// @TEST-RUN
converted := TryConvert_UDINT_TO_Destination(value, actual);
equal := actual = UDINT_TO_BOOL(value);

// @TEST-ASSERT
AssertTrue(Condition := equal, Message := 'Did not convert UDINT to BOOL correctly');
AssertTrue(Condition := converted, Message := 'Did not report UDINT to BOOL conversion was successful');

TEST_FINISHED();
END_METHOD

METHOD PUBLIC Check_UDINT_TO_BOOL_Max
VAR
	value : UDINT := DatatypeLimits.UDINT_MAX_VALUE;
	actual : BOOL;
	converted : BOOL;
	equal : BOOL;
END_VAR
TEST('Check_UDINT_TO_BOOL_Max');

// @TEST-RUN
converted := TryConvert_UDINT_TO_Destination(value, actual);
equal := actual = UDINT_TO_BOOL(value);

// @TEST-ASSERT
AssertTrue(Condition := equal, Message := 'Did not convert UDINT to BOOL correctly');
AssertTrue(Condition := converted, Message := 'Did not report UDINT to BOOL conversion was successful');

TEST_FINISHED();
END_METHOD

METHOD PUBLIC Check_UDINT_TO_BYTE_Min
VAR
	value : UDINT := DatatypeLimits.UDINT_MIN_VALUE;
	actual : BYTE;
	converted : BOOL;
	equal : BOOL;
END_VAR
TEST('Check_UDINT_TO_BYTE_Min');

// @TEST-RUN
converted := TryConvert_UDINT_TO_Destination(value, actual);
equal := actual = UDINT_TO_BYTE(value);

// @TEST-ASSERT
AssertTrue(Condition := equal, Message := 'Did not convert UDINT to BYTE correctly');
AssertTrue(Condition := converted, Message := 'Did not report UDINT to BYTE conversion was successful');

TEST_FINISHED();
END_METHOD

METHOD PUBLIC Check_UDINT_TO_BYTE_TooHigh
VAR
	value : UDINT := DatatypeLimits.UDINT_MAX_VALUE;
	actual : BYTE;
	converted : BOOL;
END_VAR
TEST('Check_UDINT_TO_BYTE_TooHigh');

// @TEST-RUN
converted := TryConvert_UDINT_TO_Destination(value, actual);

// @TEST-ASSERT
AssertFalse(Condition := converted, Message := 'Did not report UDINT to BYTE conversion was prevented');

TEST_FINISHED();
END_METHOD

METHOD PUBLIC Check_UDINT_TO_BYTE_Max
VAR
	value : UDINT := DatatypeLimits.MAX_VALUE_OF_UDINT_WHICH_CAN_BE_HELD_IN_A_BYTE;
	actual : BYTE;
	converted : BOOL;
	equal : BOOL;
END_VAR
TEST('Check_UDINT_TO_BYTE_Max');

// @TEST-RUN
converted := TryConvert_UDINT_TO_Destination(value, actual);
equal := actual = UDINT_TO_BYTE(value);

// @TEST-ASSERT
AssertTrue(Condition := equal, Message := 'Did not convert UDINT to BYTE correctly');
AssertTrue(Condition := converted, Message := 'Did not report UDINT to BYTE conversion was successful');

TEST_FINISHED();
END_METHOD

METHOD PUBLIC Check_UDINT_TO_DATE_Min
VAR
	value : UDINT := DatatypeLimits.UDINT_MIN_VALUE;
	actual : DATE;
	converted : BOOL;
	equal : BOOL;
END_VAR
TEST('Check_UDINT_TO_DATE_Min');

// @TEST-RUN
converted := TryConvert_UDINT_TO_Destination(value, actual);
equal := actual = UDINT_TO_DATE(value);

// @TEST-ASSERT
AssertTrue(Condition := equal, Message := 'Did not convert UDINT to DATE correctly');
AssertTrue(Condition := converted, Message := 'Did not report UDINT to DATE conversion was successful');

TEST_FINISHED();
END_METHOD

METHOD PUBLIC Check_UDINT_TO_DATE_Max
VAR
	value : UDINT := DatatypeLimits.UDINT_MAX_VALUE;
	actual : DATE;
	converted : BOOL;
	equal : BOOL;
END_VAR
TEST('Check_UDINT_TO_DATE_Max');

// @TEST-RUN
converted := TryConvert_UDINT_TO_Destination(value, actual);
equal := actual = UDINT_TO_DATE(value);

// @TEST-ASSERT
AssertTrue(Condition := equal, Message := 'Did not convert UDINT to DATE correctly');
AssertTrue(Condition := converted, Message := 'Did not report UDINT to DATE conversion was successful');

TEST_FINISHED();
END_METHOD

METHOD PUBLIC Check_UDINT_TO_DINT_Min
VAR
	value : UDINT := DatatypeLimits.UDINT_MIN_VALUE;
	actual : DINT;
	converted : BOOL;
	equal : BOOL;
END_VAR
TEST('Check_UDINT_TO_DINT_Min');

// @TEST-RUN
converted := TryConvert_UDINT_TO_Destination(value, actual);
equal := actual = UDINT_TO_DINT(value);

// @TEST-ASSERT
AssertTrue(Condition := equal, Message := 'Did not convert UDINT to DINT correctly');
AssertTrue(Condition := converted, Message := 'Did not report UDINT to DINT conversion was successful');

TEST_FINISHED();
END_METHOD

METHOD PUBLIC Check_UDINT_TO_DINT_TooHigh
VAR
	value : UDINT := DatatypeLimits.UDINT_MAX_VALUE;
	actual : DINT;
	converted : BOOL;
END_VAR
TEST('Check_UDINT_TO_DINT_TooHigh');

// @TEST-RUN
converted := TryConvert_UDINT_TO_Destination(value, actual);

// @TEST-ASSERT
AssertFalse(Condition := converted, Message := 'Did not report UDINT to DINT conversion was prevented');

TEST_FINISHED();
END_METHOD

METHOD PUBLIC Check_UDINT_TO_DINT_Max
VAR
	value : UDINT := DatatypeLimits.MAX_VALUE_OF_UDINT_WHICH_CAN_BE_HELD_IN_A_DINT;
	actual : DINT;
	converted : BOOL;
	equal : BOOL;
END_VAR
TEST('Check_UDINT_TO_DINT_Max');

// @TEST-RUN
converted := TryConvert_UDINT_TO_Destination(value, actual);
equal := actual = UDINT_TO_DINT(value);

// @TEST-ASSERT
AssertTrue(Condition := equal, Message := 'Did not convert UDINT to DINT correctly');
AssertTrue(Condition := converted, Message := 'Did not report UDINT to DINT conversion was successful');

TEST_FINISHED();
END_METHOD

METHOD PUBLIC Check_UDINT_TO_DT_Min
VAR
	value : UDINT := DatatypeLimits.UDINT_MIN_VALUE;
	actual : DT;
	converted : BOOL;
	equal : BOOL;
END_VAR
TEST('Check_UDINT_TO_DT_Min');

// @TEST-RUN
converted := TryConvert_UDINT_TO_Destination(value, actual);
equal := actual = UDINT_TO_DT(value);

// @TEST-ASSERT
AssertTrue(Condition := equal, Message := 'Did not convert UDINT to DT correctly');
AssertTrue(Condition := converted, Message := 'Did not report UDINT to DT conversion was successful');

TEST_FINISHED();
END_METHOD

METHOD PUBLIC Check_UDINT_TO_DT_Max
VAR
	value : UDINT := DatatypeLimits.UDINT_MAX_VALUE;
	actual : DT;
	converted : BOOL;
	equal : BOOL;
END_VAR
TEST('Check_UDINT_TO_DT_Max');

// @TEST-RUN
converted := TryConvert_UDINT_TO_Destination(value, actual);
equal := actual = UDINT_TO_DT(value);

// @TEST-ASSERT
AssertTrue(Condition := equal, Message := 'Did not convert UDINT to DT correctly');
AssertTrue(Condition := converted, Message := 'Did not report UDINT to DT conversion was successful');

TEST_FINISHED();
END_METHOD

METHOD PUBLIC Check_UDINT_TO_DWORD_Min
VAR
	value : UDINT := DatatypeLimits.UDINT_MIN_VALUE;
	actual : DWORD;
	converted : BOOL;
	equal : BOOL;
END_VAR
TEST('Check_UDINT_TO_DWORD_Min');

// @TEST-RUN
converted := TryConvert_UDINT_TO_Destination(value, actual);
equal := actual = UDINT_TO_DWORD(value);

// @TEST-ASSERT
AssertTrue(Condition := equal, Message := 'Did not convert UDINT to DWORD correctly');
AssertTrue(Condition := converted, Message := 'Did not report UDINT to DWORD conversion was successful');

TEST_FINISHED();
END_METHOD

METHOD PUBLIC Check_UDINT_TO_DWORD_Max
VAR
	value : UDINT := DatatypeLimits.UDINT_MAX_VALUE;
	actual : DWORD;
	converted : BOOL;
	equal : BOOL;
END_VAR
TEST('Check_UDINT_TO_DWORD_Max');

// @TEST-RUN
converted := TryConvert_UDINT_TO_Destination(value, actual);
equal := actual = UDINT_TO_DWORD(value);

// @TEST-ASSERT
AssertTrue(Condition := equal, Message := 'Did not convert UDINT to DWORD correctly');
AssertTrue(Condition := converted, Message := 'Did not report UDINT to DWORD conversion was successful');

TEST_FINISHED();
END_METHOD

METHOD PUBLIC Check_UDINT_TO_INT_Min
VAR
	value : UDINT := DatatypeLimits.UDINT_MIN_VALUE;
	actual : INT;
	converted : BOOL;
	equal : BOOL;
END_VAR
TEST('Check_UDINT_TO_INT_Min');

// @TEST-RUN
converted := TryConvert_UDINT_TO_Destination(value, actual);
equal := actual = UDINT_TO_INT(value);

// @TEST-ASSERT
AssertTrue(Condition := equal, Message := 'Did not convert UDINT to INT correctly');
AssertTrue(Condition := converted, Message := 'Did not report UDINT to INT conversion was successful');

TEST_FINISHED();
END_METHOD

METHOD PUBLIC Check_UDINT_TO_INT_TooHigh
VAR
	value : UDINT := DatatypeLimits.UDINT_MAX_VALUE;
	actual : INT;
	converted : BOOL;
END_VAR
TEST('Check_UDINT_TO_INT_TooHigh');

// @TEST-RUN
converted := TryConvert_UDINT_TO_Destination(value, actual);

// @TEST-ASSERT
AssertFalse(Condition := converted, Message := 'Did not report UDINT to INT conversion was prevented');

TEST_FINISHED();
END_METHOD

METHOD PUBLIC Check_UDINT_TO_INT_Max
VAR
	value : UDINT := DatatypeLimits.MAX_VALUE_OF_UDINT_WHICH_CAN_BE_HELD_IN_A_INT;
	actual : INT;
	converted : BOOL;
	equal : BOOL;
END_VAR
TEST('Check_UDINT_TO_INT_Max');

// @TEST-RUN
converted := TryConvert_UDINT_TO_Destination(value, actual);
equal := actual = UDINT_TO_INT(value);

// @TEST-ASSERT
AssertTrue(Condition := equal, Message := 'Did not convert UDINT to INT correctly');
AssertTrue(Condition := converted, Message := 'Did not report UDINT to INT conversion was successful');

TEST_FINISHED();
END_METHOD

METHOD PUBLIC Check_UDINT_TO_LINT_Min
VAR
	value : UDINT := DatatypeLimits.UDINT_MIN_VALUE;
	actual : LINT;
	converted : BOOL;
	equal : BOOL;
END_VAR
TEST('Check_UDINT_TO_LINT_Min');

// @TEST-RUN
converted := TryConvert_UDINT_TO_Destination(value, actual);
equal := actual = UDINT_TO_LINT(value);

// @TEST-ASSERT
AssertTrue(Condition := equal, Message := 'Did not convert UDINT to LINT correctly');
AssertTrue(Condition := converted, Message := 'Did not report UDINT to LINT conversion was successful');

TEST_FINISHED();
END_METHOD

METHOD PUBLIC Check_UDINT_TO_LINT_Max
VAR
	value : UDINT := DatatypeLimits.UDINT_MAX_VALUE;
	actual : LINT;
	converted : BOOL;
	equal : BOOL;
END_VAR
TEST('Check_UDINT_TO_LINT_Max');

// @TEST-RUN
converted := TryConvert_UDINT_TO_Destination(value, actual);
equal := actual = UDINT_TO_LINT(value);

// @TEST-ASSERT
AssertTrue(Condition := equal, Message := 'Did not convert UDINT to LINT correctly');
AssertTrue(Condition := converted, Message := 'Did not report UDINT to LINT conversion was successful');

TEST_FINISHED();
END_METHOD

METHOD PUBLIC Check_UDINT_TO_LREAL_Min
VAR
	value : UDINT := DatatypeLimits.UDINT_MIN_VALUE;
	actual : LREAL;
	converted : BOOL;
	equal : BOOL;
END_VAR
TEST('Check_UDINT_TO_LREAL_Min');

// @TEST-RUN
converted := TryConvert_UDINT_TO_Destination(value, actual);
equal := actual = UDINT_TO_LREAL(value);

// @TEST-ASSERT
AssertTrue(Condition := equal, Message := 'Did not convert UDINT to LREAL correctly');
AssertTrue(Condition := converted, Message := 'Did not report UDINT to LREAL conversion was successful');

TEST_FINISHED();
END_METHOD

METHOD PUBLIC Check_UDINT_TO_LREAL_Max
VAR
	value : UDINT := DatatypeLimits.UDINT_MAX_VALUE;
	actual : LREAL;
	converted : BOOL;
	equal : BOOL;
END_VAR
TEST('Check_UDINT_TO_LREAL_Max');

// @TEST-RUN
converted := TryConvert_UDINT_TO_Destination(value, actual);
equal := actual = UDINT_TO_LREAL(value);

// @TEST-ASSERT
AssertTrue(Condition := equal, Message := 'Did not convert UDINT to LREAL correctly');
AssertTrue(Condition := converted, Message := 'Did not report UDINT to LREAL conversion was successful');

TEST_FINISHED();
END_METHOD

METHOD PUBLIC Check_UDINT_TO_LWORD_Min
VAR
	value : UDINT := DatatypeLimits.UDINT_MIN_VALUE;
	actual : LWORD;
	converted : BOOL;
	equal : BOOL;
END_VAR
TEST('Check_UDINT_TO_LWORD_Min');

// @TEST-RUN
converted := TryConvert_UDINT_TO_Destination(value, actual);
equal := actual = UDINT_TO_LWORD(value);

// @TEST-ASSERT
AssertTrue(Condition := equal, Message := 'Did not convert UDINT to LWORD correctly');
AssertTrue(Condition := converted, Message := 'Did not report UDINT to LWORD conversion was successful');

TEST_FINISHED();
END_METHOD

METHOD PUBLIC Check_UDINT_TO_LWORD_Max
VAR
	value : UDINT := DatatypeLimits.UDINT_MAX_VALUE;
	actual : LWORD;
	converted : BOOL;
	equal : BOOL;
END_VAR
TEST('Check_UDINT_TO_LWORD_Max');

// @TEST-RUN
converted := TryConvert_UDINT_TO_Destination(value, actual);
equal := actual = UDINT_TO_LWORD(value);

// @TEST-ASSERT
AssertTrue(Condition := equal, Message := 'Did not convert UDINT to LWORD correctly');
AssertTrue(Condition := converted, Message := 'Did not report UDINT to LWORD conversion was successful');

TEST_FINISHED();
END_METHOD

METHOD PUBLIC Check_UDINT_TO_REAL_Min
VAR
	value : UDINT := DatatypeLimits.UDINT_MIN_VALUE;
	actual : REAL;
	converted : BOOL;
	equal : BOOL;
END_VAR
TEST('Check_UDINT_TO_REAL_Min');

// @TEST-RUN
converted := TryConvert_UDINT_TO_Destination(value, actual);
equal := actual = UDINT_TO_REAL(value);

// @TEST-ASSERT
AssertTrue(Condition := equal, Message := 'Did not convert UDINT to REAL correctly');
AssertTrue(Condition := converted, Message := 'Did not report UDINT to REAL conversion was successful');

TEST_FINISHED();
END_METHOD

METHOD PUBLIC Check_UDINT_TO_REAL_Max
VAR
	value : UDINT := DatatypeLimits.UDINT_MAX_VALUE;
	actual : REAL;
	converted : BOOL;
	equal : BOOL;
END_VAR
TEST('Check_UDINT_TO_REAL_Max');

// @TEST-RUN
converted := TryConvert_UDINT_TO_Destination(value, actual);
equal := actual = UDINT_TO_REAL(value);

// @TEST-ASSERT
AssertTrue(Condition := equal, Message := 'Did not convert UDINT to REAL correctly');
AssertTrue(Condition := converted, Message := 'Did not report UDINT to REAL conversion was successful');

TEST_FINISHED();
END_METHOD

METHOD PUBLIC Check_UDINT_TO_SINT_Min
VAR
	value : UDINT := DatatypeLimits.UDINT_MIN_VALUE;
	actual : SINT;
	converted : BOOL;
	equal : BOOL;
END_VAR
TEST('Check_UDINT_TO_SINT_Min');

// @TEST-RUN
converted := TryConvert_UDINT_TO_Destination(value, actual);
equal := actual = UDINT_TO_SINT(value);

// @TEST-ASSERT
AssertTrue(Condition := equal, Message := 'Did not convert UDINT to SINT correctly');
AssertTrue(Condition := converted, Message := 'Did not report UDINT to SINT conversion was successful');

TEST_FINISHED();
END_METHOD

METHOD PUBLIC Check_UDINT_TO_SINT_TooHigh
VAR
	value : UDINT := DatatypeLimits.UDINT_MAX_VALUE;
	actual : SINT;
	converted : BOOL;
END_VAR
TEST('Check_UDINT_TO_SINT_TooHigh');

// @TEST-RUN
converted := TryConvert_UDINT_TO_Destination(value, actual);

// @TEST-ASSERT
AssertFalse(Condition := converted, Message := 'Did not report UDINT to SINT conversion was prevented');

TEST_FINISHED();
END_METHOD

METHOD PUBLIC Check_UDINT_TO_SINT_Max
VAR
	value : UDINT := DatatypeLimits.MAX_VALUE_OF_UDINT_WHICH_CAN_BE_HELD_IN_A_SINT;
	actual : SINT;
	converted : BOOL;
	equal : BOOL;
END_VAR
TEST('Check_UDINT_TO_SINT_Max');

// @TEST-RUN
converted := TryConvert_UDINT_TO_Destination(value, actual);
equal := actual = UDINT_TO_SINT(value);

// @TEST-ASSERT
AssertTrue(Condition := equal, Message := 'Did not convert UDINT to SINT correctly');
AssertTrue(Condition := converted, Message := 'Did not report UDINT to SINT conversion was successful');

TEST_FINISHED();
END_METHOD

METHOD PUBLIC Check_UDINT_TO_STRING_Min
VAR
	value : UDINT := DatatypeLimits.UDINT_MIN_VALUE;
	actual : STRING;
	converted : BOOL;
	equal : BOOL;
END_VAR
TEST('Check_UDINT_TO_STRING_Min');

// @TEST-RUN
converted := TryConvert_UDINT_TO_Destination(value, actual);
equal := actual = UDINT_TO_STRING(value);

// @TEST-ASSERT
AssertTrue(Condition := equal, Message := 'Did not convert UDINT to STRING correctly');
AssertTrue(Condition := converted, Message := 'Did not report UDINT to STRING conversion was successful');

TEST_FINISHED();
END_METHOD

METHOD PUBLIC Check_UDINT_TO_STRING_Max
VAR
	value : UDINT := DatatypeLimits.UDINT_MAX_VALUE;
	actual : STRING;
	converted : BOOL;
	equal : BOOL;
END_VAR
TEST('Check_UDINT_TO_STRING_Max');

// @TEST-RUN
converted := TryConvert_UDINT_TO_Destination(value, actual);
equal := actual = UDINT_TO_STRING(value);

// @TEST-ASSERT
AssertTrue(Condition := equal, Message := 'Did not convert UDINT to STRING correctly');
AssertTrue(Condition := converted, Message := 'Did not report UDINT to STRING conversion was successful');

TEST_FINISHED();
END_METHOD

METHOD PUBLIC Check_UDINT_TO_TIME_Min
VAR
	value : UDINT := DatatypeLimits.UDINT_MIN_VALUE;
	actual : TIME;
	converted : BOOL;
	equal : BOOL;
END_VAR
TEST('Check_UDINT_TO_TIME_Min');

// @TEST-RUN
converted := TryConvert_UDINT_TO_Destination(value, actual);
equal := actual = UDINT_TO_TIME(value);

// @TEST-ASSERT
AssertTrue(Condition := equal, Message := 'Did not convert UDINT to TIME correctly');
AssertTrue(Condition := converted, Message := 'Did not report UDINT to TIME conversion was successful');

TEST_FINISHED();
END_METHOD

METHOD PUBLIC Check_UDINT_TO_TIME_Max
VAR
	value : UDINT := DatatypeLimits.UDINT_MAX_VALUE;
	actual : TIME;
	converted : BOOL;
	equal : BOOL;
END_VAR
TEST('Check_UDINT_TO_TIME_Max');

// @TEST-RUN
converted := TryConvert_UDINT_TO_Destination(value, actual);
equal := actual = UDINT_TO_TIME(value);

// @TEST-ASSERT
AssertTrue(Condition := equal, Message := 'Did not convert UDINT to TIME correctly');
AssertTrue(Condition := converted, Message := 'Did not report UDINT to TIME conversion was successful');

TEST_FINISHED();
END_METHOD

METHOD PUBLIC Check_UDINT_TO_TOD_Min
VAR
	value : UDINT := DatatypeLimits.UDINT_MIN_VALUE;
	actual : TOD;
	converted : BOOL;
	equal : BOOL;
END_VAR
TEST('Check_UDINT_TO_TOD_Min');

// @TEST-RUN
converted := TryConvert_UDINT_TO_Destination(value, actual);
equal := actual = UDINT_TO_TOD(value);

// @TEST-ASSERT
AssertTrue(Condition := equal, Message := 'Did not convert UDINT to TOD correctly');
AssertTrue(Condition := converted, Message := 'Did not report UDINT to TOD conversion was successful');

TEST_FINISHED();
END_METHOD

METHOD PUBLIC Check_UDINT_TO_TOD_TooHigh
VAR
	value : UDINT := DatatypeLimits.UDINT_MAX_VALUE;
	actual : TOD;
	converted : BOOL;
END_VAR
TEST('Check_UDINT_TO_TOD_TooHigh');

// @TEST-RUN
converted := TryConvert_UDINT_TO_Destination(value, actual);

// @TEST-ASSERT
AssertFalse(Condition := converted, Message := 'Did not report UDINT to TOD conversion was prevented');

TEST_FINISHED();
END_METHOD

METHOD PUBLIC Check_UDINT_TO_TOD_Max
VAR
	value : UDINT := DatatypeLimits.MAX_VALUE_OF_UDINT_WHICH_CAN_BE_HELD_IN_A_TOD;
	actual : TOD;
	converted : BOOL;
	equal : BOOL;
END_VAR
TEST('Check_UDINT_TO_TOD_Max');

// @TEST-RUN
converted := TryConvert_UDINT_TO_Destination(value, actual);
equal := actual = UDINT_TO_TOD(value);

// @TEST-ASSERT
AssertTrue(Condition := equal, Message := 'Did not convert UDINT to TOD correctly');
AssertTrue(Condition := converted, Message := 'Did not report UDINT to TOD conversion was successful');

TEST_FINISHED();
END_METHOD

METHOD PUBLIC Check_UDINT_TO_UDINT_Min
VAR
	value : UDINT := DatatypeLimits.UDINT_MIN_VALUE;
	actual : UDINT;
	converted : BOOL;
	equal : BOOL;
END_VAR
TEST('Check_UDINT_TO_UDINT_Min');

// @TEST-RUN
converted := TryConvert_UDINT_TO_Destination(value, actual);
equal := actual = value;

// @TEST-ASSERT
AssertTrue(Condition := equal, Message := 'Did not convert UDINT to UDINT correctly');
AssertTrue(Condition := converted, Message := 'Did not report UDINT to UDINT conversion was successful');

TEST_FINISHED();
END_METHOD

METHOD PUBLIC Check_UDINT_TO_UDINT_Max
VAR
	value : UDINT := DatatypeLimits.UDINT_MAX_VALUE;
	actual : UDINT;
	converted : BOOL;
	equal : BOOL;
END_VAR
TEST('Check_UDINT_TO_UDINT_Max');

// @TEST-RUN
converted := TryConvert_UDINT_TO_Destination(value, actual);
equal := actual = value;

// @TEST-ASSERT
AssertTrue(Condition := equal, Message := 'Did not convert UDINT to UDINT correctly');
AssertTrue(Condition := converted, Message := 'Did not report UDINT to UDINT conversion was successful');

TEST_FINISHED();
END_METHOD

METHOD PUBLIC Check_UDINT_TO_UINT_Min
VAR
	value : UDINT := DatatypeLimits.UDINT_MIN_VALUE;
	actual : UINT;
	converted : BOOL;
	equal : BOOL;
END_VAR
TEST('Check_UDINT_TO_UINT_Min');

// @TEST-RUN
converted := TryConvert_UDINT_TO_Destination(value, actual);
equal := actual = UDINT_TO_UINT(value);

// @TEST-ASSERT
AssertTrue(Condition := equal, Message := 'Did not convert UDINT to UINT correctly');
AssertTrue(Condition := converted, Message := 'Did not report UDINT to UINT conversion was successful');

TEST_FINISHED();
END_METHOD

METHOD PUBLIC Check_UDINT_TO_UINT_TooHigh
VAR
	value : UDINT := DatatypeLimits.UDINT_MAX_VALUE;
	actual : UINT;
	converted : BOOL;
END_VAR
TEST('Check_UDINT_TO_UINT_TooHigh');

// @TEST-RUN
converted := TryConvert_UDINT_TO_Destination(value, actual);

// @TEST-ASSERT
AssertFalse(Condition := converted, Message := 'Did not report UDINT to UINT conversion was prevented');

TEST_FINISHED();
END_METHOD

METHOD PUBLIC Check_UDINT_TO_UINT_Max
VAR
	value : UDINT := DatatypeLimits.MAX_VALUE_OF_UDINT_WHICH_CAN_BE_HELD_IN_A_UINT;
	actual : UINT;
	converted : BOOL;
	equal : BOOL;
END_VAR
TEST('Check_UDINT_TO_UINT_Max');

// @TEST-RUN
converted := TryConvert_UDINT_TO_Destination(value, actual);
equal := actual = UDINT_TO_UINT(value);

// @TEST-ASSERT
AssertTrue(Condition := equal, Message := 'Did not convert UDINT to UINT correctly');
AssertTrue(Condition := converted, Message := 'Did not report UDINT to UINT conversion was successful');

TEST_FINISHED();
END_METHOD

METHOD PUBLIC Check_UDINT_TO_ULINT_Min
VAR
	value : UDINT := DatatypeLimits.UDINT_MIN_VALUE;
	actual : ULINT;
	converted : BOOL;
	equal : BOOL;
END_VAR
TEST('Check_UDINT_TO_ULINT_Min');

// @TEST-RUN
converted := TryConvert_UDINT_TO_Destination(value, actual);
equal := actual = UDINT_TO_ULINT(value);

// @TEST-ASSERT
AssertTrue(Condition := equal, Message := 'Did not convert UDINT to ULINT correctly');
AssertTrue(Condition := converted, Message := 'Did not report UDINT to ULINT conversion was successful');

TEST_FINISHED();
END_METHOD

METHOD PUBLIC Check_UDINT_TO_ULINT_Max
VAR
	value : UDINT := DatatypeLimits.UDINT_MAX_VALUE;
	actual : ULINT;
	converted : BOOL;
	equal : BOOL;
END_VAR
TEST('Check_UDINT_TO_ULINT_Max');

// @TEST-RUN
converted := TryConvert_UDINT_TO_Destination(value, actual);
equal := actual = UDINT_TO_ULINT(value);

// @TEST-ASSERT
AssertTrue(Condition := equal, Message := 'Did not convert UDINT to ULINT correctly');
AssertTrue(Condition := converted, Message := 'Did not report UDINT to ULINT conversion was successful');

TEST_FINISHED();
END_METHOD

METHOD PUBLIC Check_UDINT_TO_USINT_Min
VAR
	value : UDINT := DatatypeLimits.UDINT_MIN_VALUE;
	actual : USINT;
	converted : BOOL;
	equal : BOOL;
END_VAR
TEST('Check_UDINT_TO_USINT_Min');

// @TEST-RUN
converted := TryConvert_UDINT_TO_Destination(value, actual);
equal := actual = UDINT_TO_USINT(value);

// @TEST-ASSERT
AssertTrue(Condition := equal, Message := 'Did not convert UDINT to USINT correctly');
AssertTrue(Condition := converted, Message := 'Did not report UDINT to USINT conversion was successful');

TEST_FINISHED();
END_METHOD

METHOD PUBLIC Check_UDINT_TO_USINT_TooHigh
VAR
	value : UDINT := DatatypeLimits.UDINT_MAX_VALUE;
	actual : USINT;
	converted : BOOL;
END_VAR
TEST('Check_UDINT_TO_USINT_TooHigh');

// @TEST-RUN
converted := TryConvert_UDINT_TO_Destination(value, actual);

// @TEST-ASSERT
AssertFalse(Condition := converted, Message := 'Did not report UDINT to USINT conversion was prevented');

TEST_FINISHED();
END_METHOD

METHOD PUBLIC Check_UDINT_TO_USINT_Max
VAR
	value : UDINT := DatatypeLimits.MAX_VALUE_OF_UDINT_WHICH_CAN_BE_HELD_IN_A_USINT;
	actual : USINT;
	converted : BOOL;
	equal : BOOL;
END_VAR
TEST('Check_UDINT_TO_USINT_Max');

// @TEST-RUN
converted := TryConvert_UDINT_TO_Destination(value, actual);
equal := actual = UDINT_TO_USINT(value);

// @TEST-ASSERT
AssertTrue(Condition := equal, Message := 'Did not convert UDINT to USINT correctly');
AssertTrue(Condition := converted, Message := 'Did not report UDINT to USINT conversion was successful');

TEST_FINISHED();
END_METHOD

METHOD PUBLIC Check_UDINT_TO_WORD_Min
VAR
	value : UDINT := DatatypeLimits.UDINT_MIN_VALUE;
	actual : WORD;
	converted : BOOL;
	equal : BOOL;
END_VAR
TEST('Check_UDINT_TO_WORD_Min');

// @TEST-RUN
converted := TryConvert_UDINT_TO_Destination(value, actual);
equal := actual = UDINT_TO_WORD(value);

// @TEST-ASSERT
AssertTrue(Condition := equal, Message := 'Did not convert UDINT to WORD correctly');
AssertTrue(Condition := converted, Message := 'Did not report UDINT to WORD conversion was successful');

TEST_FINISHED();
END_METHOD

METHOD PUBLIC Check_UDINT_TO_WORD_TooHigh
VAR
	value : UDINT := DatatypeLimits.UDINT_MAX_VALUE;
	actual : WORD;
	converted : BOOL;
END_VAR
TEST('Check_UDINT_TO_WORD_TooHigh');

// @TEST-RUN
converted := TryConvert_UDINT_TO_Destination(value, actual);

// @TEST-ASSERT
AssertFalse(Condition := converted, Message := 'Did not report UDINT to WORD conversion was prevented');

TEST_FINISHED();
END_METHOD

METHOD PUBLIC Check_UDINT_TO_WORD_Max
VAR
	value : UDINT := DatatypeLimits.MAX_VALUE_OF_UDINT_WHICH_CAN_BE_HELD_IN_A_WORD;
	actual : WORD;
	converted : BOOL;
	equal : BOOL;
END_VAR
TEST('Check_UDINT_TO_WORD_Max');

// @TEST-RUN
converted := TryConvert_UDINT_TO_Destination(value, actual);
equal := actual = UDINT_TO_WORD(value);

// @TEST-ASSERT
AssertTrue(Condition := equal, Message := 'Did not convert UDINT to WORD correctly');
AssertTrue(Condition := converted, Message := 'Did not report UDINT to WORD conversion was successful');

TEST_FINISHED();
END_METHOD

END_FUNCTION_BLOCK

// ---- Tests/ULINT_TO_TestSuite.TcPOU
FUNCTION_BLOCK PUBLIC ULINT_TO_TestSuite EXTENDS TcUnit.FB_TestSuite
VAR
END_VAR

Check_ULINT_TO_BOOL_Max();
Check_ULINT_TO_BOOL_Min();
Check_ULINT_TO_BYTE_Max();
Check_ULINT_TO_BYTE_Min();
Check_ULINT_TO_BYTE_TooHigh();
Check_ULINT_TO_WORD_Max();
Check_ULINT_TO_WORD_Min();
Check_ULINT_TO_WORD_TooHigh();
Check_ULINT_TO_DWORD_Max();
Check_ULINT_TO_DWORD_Min();
Check_ULINT_TO_DWORD_TooHigh();
Check_ULINT_TO_LWORD_Max();
Check_ULINT_TO_LWORD_Min();
Check_ULINT_TO_SINT_Max();
Check_ULINT_TO_SINT_Min();
Check_ULINT_TO_SINT_TooHigh();
Check_ULINT_TO_INT_Max();
Check_ULINT_TO_INT_Min();
Check_ULINT_TO_INT_TooHigh();
Check_ULINT_TO_DINT_Max();
Check_ULINT_TO_DINT_Min();
Check_ULINT_TO_DINT_TooHigh();
Check_ULINT_TO_LINT_Max();
Check_ULINT_TO_LINT_Min();
Check_ULINT_TO_LINT_TooHigh();
Check_ULINT_TO_USINT_Max();
Check_ULINT_TO_USINT_Min();
Check_ULINT_TO_USINT_TooHigh();
Check_ULINT_TO_UINT_Max();
Check_ULINT_TO_UINT_Min();
Check_ULINT_TO_UINT_TooHigh();
Check_ULINT_TO_UDINT_Max();
Check_ULINT_TO_UDINT_Min();
Check_ULINT_TO_UDINT_TooHigh();
Check_ULINT_TO_ULINT_Max();
Check_ULINT_TO_ULINT_Min();
Check_ULINT_TO_REAL_Max();
Check_ULINT_TO_REAL_Min();
Check_ULINT_TO_LREAL_Max();
Check_ULINT_TO_LREAL_Min();
Check_ULINT_TO_TIME_Max();
Check_ULINT_TO_TIME_Min();
Check_ULINT_TO_TIME_TooHigh();
Check_ULINT_TO_TOD_Max();
Check_ULINT_TO_TOD_Min();
Check_ULINT_TO_TOD_TooHigh();
Check_ULINT_TO_DATE_Max();
Check_ULINT_TO_DATE_Min();
Check_ULINT_TO_DATE_TooHigh();
Check_ULINT_TO_DT_Max();
Check_ULINT_TO_DT_Min();
Check_ULINT_TO_DT_TooHigh();
Check_ULINT_TO_STRING_Max();
Check_ULINT_TO_STRING_Min();

METHOD PUBLIC Check_ULINT_TO_BOOL_Min
VAR
	value : ULINT := DatatypeLimits.ULINT_MIN_VALUE;
	actual : BOOL;
	converted : BOOL;
	equal : BOOL;
END_VAR
TEST('Check_ULINT_TO_BOOL_Min');

// @TEST-RUN
converted := TryConvert_ULINT_TO_Destination(value, actual);
equal := actual = ULINT_TO_BOOL(value);

// @TEST-ASSERT
AssertTrue(Condition := equal, Message := 'Did not convert ULINT to BOOL correctly');
AssertTrue(Condition := converted, Message := 'Did not report ULINT to BOOL conversion was successful');

TEST_FINISHED();
END_METHOD

METHOD PUBLIC Check_ULINT_TO_BOOL_Max
VAR
	value : ULINT := DatatypeLimits.ULINT_MAX_VALUE;
	actual : BOOL;
	converted : BOOL;
	equal : BOOL;
END_VAR
TEST('Check_ULINT_TO_BOOL_Max');

// @TEST-RUN
converted := TryConvert_ULINT_TO_Destination(value, actual);
equal := actual = ULINT_TO_BOOL(value);

// @TEST-ASSERT
AssertTrue(Condition := equal, Message := 'Did not convert ULINT to BOOL correctly');
AssertTrue(Condition := converted, Message := 'Did not report ULINT to BOOL conversion was successful');

TEST_FINISHED();
END_METHOD

METHOD PUBLIC Check_ULINT_TO_BYTE_Min
VAR
	value : ULINT := DatatypeLimits.ULINT_MIN_VALUE;
	actual : BYTE;
	converted : BOOL;
	equal : BOOL;
END_VAR
TEST('Check_ULINT_TO_BYTE_Min');

// @TEST-RUN
converted := TryConvert_ULINT_TO_Destination(value, actual);
equal := actual = ULINT_TO_BYTE(value);

// @TEST-ASSERT
AssertTrue(Condition := equal, Message := 'Did not convert ULINT to BYTE correctly');
AssertTrue(Condition := converted, Message := 'Did not report ULINT to BYTE conversion was successful');

TEST_FINISHED();
END_METHOD

METHOD PUBLIC Check_ULINT_TO_BYTE_TooHigh
VAR
	value : ULINT := DatatypeLimits.ULINT_MAX_VALUE;
	actual : BYTE;
	converted : BOOL;
END_VAR
TEST('Check_ULINT_TO_BYTE_TooHigh');

// @TEST-RUN
converted := TryConvert_ULINT_TO_Destination(value, actual);

// @TEST-ASSERT
AssertFalse(Condition := converted, Message := 'Did not report ULINT to BYTE conversion was prevented');

TEST_FINISHED();
END_METHOD

METHOD PUBLIC Check_ULINT_TO_BYTE_Max
VAR
	value : ULINT := DatatypeLimits.MAX_VALUE_OF_ULINT_WHICH_CAN_BE_HELD_IN_A_BYTE;
	actual : BYTE;
	converted : BOOL;
	equal : BOOL;
END_VAR
TEST('Check_ULINT_TO_BYTE_Max');

// @TEST-RUN
converted := TryConvert_ULINT_TO_Destination(value, actual);
equal := actual = ULINT_TO_BYTE(value);

// @TEST-ASSERT
AssertTrue(Condition := equal, Message := 'Did not convert ULINT to BYTE correctly');
AssertTrue(Condition := converted, Message := 'Did not report ULINT to BYTE conversion was successful');

TEST_FINISHED();
END_METHOD

METHOD PUBLIC Check_ULINT_TO_DATE_Min
VAR
	value : ULINT := DatatypeLimits.ULINT_MIN_VALUE;
	actual : DATE;
	converted : BOOL;
	equal : BOOL;
END_VAR
TEST('Check_ULINT_TO_DATE_Min');

// @TEST-RUN
converted := TryConvert_ULINT_TO_Destination(value, actual);
equal := actual = ULINT_TO_DATE(value);

// @TEST-ASSERT
AssertTrue(Condition := equal, Message := 'Did not convert ULINT to DATE correctly');
AssertTrue(Condition := converted, Message := 'Did not report ULINT to DATE conversion was successful');

TEST_FINISHED();
END_METHOD

METHOD PUBLIC Check_ULINT_TO_DATE_TooHigh
VAR
	value : ULINT := DatatypeLimits.ULINT_MAX_VALUE;
	actual : DATE;
	converted : BOOL;
END_VAR
TEST('Check_ULINT_TO_DATE_TooHigh');

// @TEST-RUN
converted := TryConvert_ULINT_TO_Destination(value, actual);

// @TEST-ASSERT
AssertFalse(Condition := converted, Message := 'Did not report ULINT to DATE conversion was prevented');

TEST_FINISHED();
END_METHOD

METHOD PUBLIC Check_ULINT_TO_DATE_Max
VAR
	value : ULINT := DatatypeLimits.MAX_VALUE_OF_ULINT_WHICH_CAN_BE_HELD_IN_A_DATE;
	actual : DATE;
	converted : BOOL;
	equal : BOOL;
END_VAR
TEST('Check_ULINT_TO_DATE_Max');

// @TEST-RUN
converted := TryConvert_ULINT_TO_Destination(value, actual);
equal := actual = ULINT_TO_DATE(value);

// @TEST-ASSERT
AssertTrue(Condition := equal, Message := 'Did not convert ULINT to DATE correctly');
AssertTrue(Condition := converted, Message := 'Did not report ULINT to DATE conversion was successful');

TEST_FINISHED();
END_METHOD

METHOD PUBLIC Check_ULINT_TO_DINT_Min
VAR
	value : ULINT := DatatypeLimits.ULINT_MIN_VALUE;
	actual : DINT;
	converted : BOOL;
	equal : BOOL;
END_VAR
TEST('Check_ULINT_TO_DINT_Min');

// @TEST-RUN
converted := TryConvert_ULINT_TO_Destination(value, actual);
equal := actual = ULINT_TO_DINT(value);

// @TEST-ASSERT
AssertTrue(Condition := equal, Message := 'Did not convert ULINT to DINT correctly');
AssertTrue(Condition := converted, Message := 'Did not report ULINT to DINT conversion was successful');

TEST_FINISHED();
END_METHOD

METHOD PUBLIC Check_ULINT_TO_DINT_TooHigh
VAR
	value : ULINT := DatatypeLimits.ULINT_MAX_VALUE;
	actual : DINT;
	converted : BOOL;
END_VAR
TEST('Check_ULINT_TO_DINT_TooHigh');

// @TEST-RUN
converted := TryConvert_ULINT_TO_Destination(value, actual);

// @TEST-ASSERT
AssertFalse(Condition := converted, Message := 'Did not report ULINT to DINT conversion was prevented');

TEST_FINISHED();
END_METHOD

METHOD PUBLIC Check_ULINT_TO_DINT_Max
VAR
	value : ULINT := DatatypeLimits.MAX_VALUE_OF_ULINT_WHICH_CAN_BE_HELD_IN_A_DINT;
	actual : DINT;
	converted : BOOL;
	equal : BOOL;
END_VAR
TEST('Check_ULINT_TO_DINT_Max');

// @TEST-RUN
converted := TryConvert_ULINT_TO_Destination(value, actual);
equal := actual = ULINT_TO_DINT(value);

// @TEST-ASSERT
AssertTrue(Condition := equal, Message := 'Did not convert ULINT to DINT correctly');
AssertTrue(Condition := converted, Message := 'Did not report ULINT to DINT conversion was successful');

TEST_FINISHED();
END_METHOD

METHOD PUBLIC Check_ULINT_TO_DT_Min
VAR
	value : ULINT := DatatypeLimits.ULINT_MIN_VALUE;
	actual : DT;
	converted : BOOL;
	equal : BOOL;
END_VAR
TEST('Check_ULINT_TO_DT_Min');

// @TEST-RUN
converted := TryConvert_ULINT_TO_Destination(value, actual);
equal := actual = ULINT_TO_DT(value);

// @TEST-ASSERT
AssertTrue(Condition := equal, Message := 'Did not convert ULINT to DT correctly');
AssertTrue(Condition := converted, Message := 'Did not report ULINT to DT conversion was successful');

TEST_FINISHED();
END_METHOD

METHOD PUBLIC Check_ULINT_TO_DT_TooHigh
VAR
	value : ULINT := DatatypeLimits.ULINT_MAX_VALUE;
	actual : DT;
	converted : BOOL;
END_VAR
TEST('Check_ULINT_TO_DT_TooHigh');

// @TEST-RUN
converted := TryConvert_ULINT_TO_Destination(value, actual);

// @TEST-ASSERT
AssertFalse(Condition := converted, Message := 'Did not report ULINT to DT conversion was prevented');

TEST_FINISHED();
END_METHOD

METHOD PUBLIC Check_ULINT_TO_DT_Max
VAR
	value : ULINT := DatatypeLimits.MAX_VALUE_OF_ULINT_WHICH_CAN_BE_HELD_IN_A_DT;
	actual : DT;
	converted : BOOL;
	equal : BOOL;
END_VAR
TEST('Check_ULINT_TO_DT_Max');

// @TEST-RUN
converted := TryConvert_ULINT_TO_Destination(value, actual);
equal := actual = ULINT_TO_DT(value);

// @TEST-ASSERT
AssertTrue(Condition := equal, Message := 'Did not convert ULINT to DT correctly');
AssertTrue(Condition := converted, Message := 'Did not report ULINT to DT conversion was successful');

TEST_FINISHED();
END_METHOD

METHOD PUBLIC Check_ULINT_TO_DWORD_Min
VAR
	value : ULINT := DatatypeLimits.ULINT_MIN_VALUE;
	actual : DWORD;
	converted : BOOL;
	equal : BOOL;
END_VAR
TEST('Check_ULINT_TO_DWORD_Min');

// @TEST-RUN
converted := TryConvert_ULINT_TO_Destination(value, actual);
equal := actual = ULINT_TO_DWORD(value);

// @TEST-ASSERT
AssertTrue(Condition := equal, Message := 'Did not convert ULINT to DWORD correctly');
AssertTrue(Condition := converted, Message := 'Did not report ULINT to DWORD conversion was successful');

TEST_FINISHED();
END_METHOD

METHOD PUBLIC Check_ULINT_TO_DWORD_TooHigh
VAR
	value : ULINT := DatatypeLimits.ULINT_MAX_VALUE;
	actual : DWORD;
	converted : BOOL;
END_VAR
TEST('Check_ULINT_TO_DWORD_TooHigh');

// @TEST-RUN
converted := TryConvert_ULINT_TO_Destination(value, actual);

// @TEST-ASSERT
AssertFalse(Condition := converted, Message := 'Did not report ULINT to DWORD conversion was prevented');

TEST_FINISHED();
END_METHOD

METHOD PUBLIC Check_ULINT_TO_DWORD_Max
VAR
	value : ULINT := DatatypeLimits.MAX_VALUE_OF_ULINT_WHICH_CAN_BE_HELD_IN_A_DWORD;
	actual : DWORD;
	converted : BOOL;
	equal : BOOL;
END_VAR
TEST('Check_ULINT_TO_DWORD_Max');

// @TEST-RUN
converted := TryConvert_ULINT_TO_Destination(value, actual);
equal := actual = ULINT_TO_DWORD(value);

// @TEST-ASSERT
AssertTrue(Condition := equal, Message := 'Did not convert ULINT to DWORD correctly');
AssertTrue(Condition := converted, Message := 'Did not report ULINT to DWORD conversion was successful');

TEST_FINISHED();
END_METHOD

METHOD PUBLIC Check_ULINT_TO_INT_Min
VAR
	value : ULINT := DatatypeLimits.ULINT_MIN_VALUE;
	actual : INT;
	converted : BOOL;
	equal : BOOL;
END_VAR
TEST('Check_ULINT_TO_INT_Min');

// @TEST-RUN
converted := TryConvert_ULINT_TO_Destination(value, actual);
equal := actual = ULINT_TO_INT(value);

// @TEST-ASSERT
AssertTrue(Condition := equal, Message := 'Did not convert ULINT to INT correctly');
AssertTrue(Condition := converted, Message := 'Did not report ULINT to INT conversion was successful');

TEST_FINISHED();
END_METHOD

METHOD PUBLIC Check_ULINT_TO_INT_TooHigh
VAR
	value : ULINT := DatatypeLimits.ULINT_MAX_VALUE;
	actual : INT;
	converted : BOOL;
END_VAR
TEST('Check_ULINT_TO_INT_TooHigh');

// @TEST-RUN
converted := TryConvert_ULINT_TO_Destination(value, actual);

// @TEST-ASSERT
AssertFalse(Condition := converted, Message := 'Did not report ULINT to INT conversion was prevented');

TEST_FINISHED();
END_METHOD

METHOD PUBLIC Check_ULINT_TO_INT_Max
VAR
	value : ULINT := DatatypeLimits.MAX_VALUE_OF_ULINT_WHICH_CAN_BE_HELD_IN_A_INT;
	actual : INT;
	converted : BOOL;
	equal : BOOL;
END_VAR
TEST('Check_ULINT_TO_INT_Max');

// @TEST-RUN
converted := TryConvert_ULINT_TO_Destination(value, actual);
equal := actual = ULINT_TO_INT(value);

// @TEST-ASSERT
AssertTrue(Condition := equal, Message := 'Did not convert ULINT to INT correctly');
AssertTrue(Condition := converted, Message := 'Did not report ULINT to INT conversion was successful');

TEST_FINISHED();
END_METHOD

METHOD PUBLIC Check_ULINT_TO_LINT_Min
VAR
	value : ULINT := DatatypeLimits.ULINT_MIN_VALUE;
	actual : LINT;
	converted : BOOL;
	equal : BOOL;
END_VAR
TEST('Check_ULINT_TO_LINT_Min');

// @TEST-RUN
converted := TryConvert_ULINT_TO_Destination(value, actual);
equal := actual = ULINT_TO_LINT(value);

// @TEST-ASSERT
AssertTrue(Condition := equal, Message := 'Did not convert ULINT to LINT correctly');
AssertTrue(Condition := converted, Message := 'Did not report ULINT to LINT conversion was successful');

TEST_FINISHED();
END_METHOD

METHOD PUBLIC Check_ULINT_TO_LINT_TooHigh
VAR
	value : ULINT := DatatypeLimits.ULINT_MAX_VALUE;
	actual : LINT;
	converted : BOOL;
END_VAR
TEST('Check_ULINT_TO_LINT_TooHigh');

// @TEST-RUN
converted := TryConvert_ULINT_TO_Destination(value, actual);

// @TEST-ASSERT
AssertFalse(Condition := converted, Message := 'Did not report ULINT to LINT conversion was prevented');

TEST_FINISHED();
END_METHOD

METHOD PUBLIC Check_ULINT_TO_LINT_Max
VAR
	value : ULINT := DatatypeLimits.MAX_VALUE_OF_ULINT_WHICH_CAN_BE_HELD_IN_A_LINT;
	actual : LINT;
	converted : BOOL;
	equal : BOOL;
END_VAR
TEST('Check_ULINT_TO_LINT_Max');

// @TEST-RUN
converted := TryConvert_ULINT_TO_Destination(value, actual);
equal := actual = ULINT_TO_LINT(value);

// @TEST-ASSERT
AssertTrue(Condition := equal, Message := 'Did not convert ULINT to LINT correctly');
AssertTrue(Condition := converted, Message := 'Did not report ULINT to LINT conversion was successful');

TEST_FINISHED();
END_METHOD

METHOD PUBLIC Check_ULINT_TO_LREAL_Min
VAR
	value : ULINT := DatatypeLimits.ULINT_MIN_VALUE;
	actual : LREAL;
	converted : BOOL;
	equal : BOOL;
END_VAR
TEST('Check_ULINT_TO_LREAL_Min');

// @TEST-RUN
converted := TryConvert_ULINT_TO_Destination(value, actual);
equal := actual = ULINT_TO_LREAL(value);

// @TEST-ASSERT
AssertTrue(Condition := equal, Message := 'Did not convert ULINT to LREAL correctly');
AssertTrue(Condition := converted, Message := 'Did not report ULINT to LREAL conversion was successful');

TEST_FINISHED();
END_METHOD

METHOD PUBLIC Check_ULINT_TO_LREAL_Max
VAR
	value : ULINT := DatatypeLimits.ULINT_MAX_VALUE;
	actual : LREAL;
	converted : BOOL;
	equal : BOOL;
END_VAR
TEST('Check_ULINT_TO_LREAL_Max');

// @TEST-RUN
converted := TryConvert_ULINT_TO_Destination(value, actual);
equal := actual = ULINT_TO_LREAL(value);

// @TEST-ASSERT
AssertTrue(Condition := equal, Message := 'Did not convert ULINT to LREAL correctly');
AssertTrue(Condition := converted, Message := 'Did not report ULINT to LREAL conversion was successful');

TEST_FINISHED();
END_METHOD

METHOD PUBLIC Check_ULINT_TO_LWORD_Min
VAR
	value : ULINT := DatatypeLimits.ULINT_MIN_VALUE;
	actual : LWORD;
	converted : BOOL;
	equal : BOOL;
END_VAR
TEST('Check_ULINT_TO_LWORD_Min');

// @TEST-RUN
converted := TryConvert_ULINT_TO_Destination(value, actual);
equal := actual = ULINT_TO_LWORD(value);

// @TEST-ASSERT
AssertTrue(Condition := equal, Message := 'Did not convert ULINT to LWORD correctly');
AssertTrue(Condition := converted, Message := 'Did not report ULINT to LWORD conversion was successful');

TEST_FINISHED();
END_METHOD

METHOD PUBLIC Check_ULINT_TO_LWORD_Max
VAR
	value : ULINT := DatatypeLimits.ULINT_MAX_VALUE;
	actual : LWORD;
	converted : BOOL;
	equal : BOOL;
END_VAR
TEST('Check_ULINT_TO_LWORD_Max');

// @TEST-RUN
converted := TryConvert_ULINT_TO_Destination(value, actual);
equal := actual = ULINT_TO_LWORD(value);

// @TEST-ASSERT
AssertTrue(Condition := equal, Message := 'Did not convert ULINT to LWORD correctly');
AssertTrue(Condition := converted, Message := 'Did not report ULINT to LWORD conversion was successful');

TEST_FINISHED();
END_METHOD

METHOD PUBLIC Check_ULINT_TO_REAL_Min
VAR
	value : ULINT := DatatypeLimits.ULINT_MIN_VALUE;
	actual : REAL;
	converted : BOOL;
	equal : BOOL;
END_VAR
TEST('Check_ULINT_TO_REAL_Min');

// @TEST-RUN
converted := TryConvert_ULINT_TO_Destination(value, actual);
equal := actual = ULINT_TO_REAL(value);

// @TEST-ASSERT
AssertTrue(Condition := equal, Message := 'Did not convert ULINT to REAL correctly');
AssertTrue(Condition := converted, Message := 'Did not report ULINT to REAL conversion was successful');

TEST_FINISHED();
END_METHOD

METHOD PUBLIC Check_ULINT_TO_REAL_Max
VAR
	value : ULINT := DatatypeLimits.ULINT_MAX_VALUE;
	actual : REAL;
	converted : BOOL;
	equal : BOOL;
END_VAR
TEST('Check_ULINT_TO_REAL_Max');

// @TEST-RUN
converted := TryConvert_ULINT_TO_Destination(value, actual);
equal := actual = ULINT_TO_REAL(value);

// @TEST-ASSERT
AssertTrue(Condition := equal, Message := 'Did not convert ULINT to REAL correctly');
AssertTrue(Condition := converted, Message := 'Did not report ULINT to REAL conversion was successful');

TEST_FINISHED();
END_METHOD

METHOD PUBLIC Check_ULINT_TO_SINT_Min
VAR
	value : ULINT := DatatypeLimits.ULINT_MIN_VALUE;
	actual : SINT;
	converted : BOOL;
	equal : BOOL;
END_VAR
TEST('Check_ULINT_TO_SINT_Min');

// @TEST-RUN
converted := TryConvert_ULINT_TO_Destination(value, actual);
equal := actual = ULINT_TO_SINT(value);

// @TEST-ASSERT
AssertTrue(Condition := equal, Message := 'Did not convert ULINT to SINT correctly');
AssertTrue(Condition := converted, Message := 'Did not report ULINT to SINT conversion was successful');

TEST_FINISHED();
END_METHOD

METHOD PUBLIC Check_ULINT_TO_SINT_TooHigh
VAR
	value : ULINT := DatatypeLimits.ULINT_MAX_VALUE;
	actual : SINT;
	converted : BOOL;
END_VAR
TEST('Check_ULINT_TO_SINT_TooHigh');

// @TEST-RUN
converted := TryConvert_ULINT_TO_Destination(value, actual);

// @TEST-ASSERT
AssertFalse(Condition := converted, Message := 'Did not report ULINT to SINT conversion was prevented');

TEST_FINISHED();
END_METHOD

METHOD PUBLIC Check_ULINT_TO_SINT_Max
VAR
	value : ULINT := DatatypeLimits.MAX_VALUE_OF_ULINT_WHICH_CAN_BE_HELD_IN_A_SINT;
	actual : SINT;
	converted : BOOL;
	equal : BOOL;
END_VAR
TEST('Check_ULINT_TO_SINT_Max');

// @TEST-RUN
converted := TryConvert_ULINT_TO_Destination(value, actual);
equal := actual = ULINT_TO_SINT(value);

// @TEST-ASSERT
AssertTrue(Condition := equal, Message := 'Did not convert ULINT to SINT correctly');
AssertTrue(Condition := converted, Message := 'Did not report ULINT to SINT conversion was successful');

TEST_FINISHED();
END_METHOD

METHOD PUBLIC Check_ULINT_TO_STRING_Min
VAR
	value : ULINT := DatatypeLimits.ULINT_MIN_VALUE;
	actual : STRING;
	converted : BOOL;
	equal : BOOL;
END_VAR
TEST('Check_ULINT_TO_STRING_Min');

// @TEST-RUN
converted := TryConvert_ULINT_TO_Destination(value, actual);
equal := actual = ULINT_TO_STRING(value);

// @TEST-ASSERT
AssertTrue(Condition := equal, Message := 'Did not convert ULINT to STRING correctly');
AssertTrue(Condition := converted, Message := 'Did not report ULINT to STRING conversion was successful');

TEST_FINISHED();
END_METHOD

METHOD PUBLIC Check_ULINT_TO_STRING_Max
VAR
	value : ULINT := DatatypeLimits.ULINT_MAX_VALUE;
	actual : STRING;
	converted : BOOL;
	equal : BOOL;
END_VAR
TEST('Check_ULINT_TO_STRING_Max');

// @TEST-RUN
converted := TryConvert_ULINT_TO_Destination(value, actual);
equal := actual = ULINT_TO_STRING(value);

// @TEST-ASSERT
AssertTrue(Condition := equal, Message := 'Did not convert ULINT to STRING correctly');
AssertTrue(Condition := converted, Message := 'Did not report ULINT to STRING conversion was successful');

TEST_FINISHED();
END_METHOD

METHOD PUBLIC Check_ULINT_TO_TIME_Min
VAR
	value : ULINT := DatatypeLimits.ULINT_MIN_VALUE;
	actual : TIME;
	converted : BOOL;
	equal : BOOL;
END_VAR
TEST('Check_ULINT_TO_TIME_Min');

// @TEST-RUN
converted := TryConvert_ULINT_TO_Destination(value, actual);
equal := actual = ULINT_TO_TIME(value);

// @TEST-ASSERT
AssertTrue(Condition := equal, Message := 'Did not convert ULINT to TIME correctly');
AssertTrue(Condition := converted, Message := 'Did not report ULINT to TIME conversion was successful');

TEST_FINISHED();
END_METHOD

METHOD PUBLIC Check_ULINT_TO_TIME_TooHigh
VAR
	value : ULINT := DatatypeLimits.ULINT_MAX_VALUE;
	actual : TIME;
	converted : BOOL;
END_VAR
TEST('Check_ULINT_TO_TIME_TooHigh');

// @TEST-RUN
converted := TryConvert_ULINT_TO_Destination(value, actual);

// @TEST-ASSERT
AssertFalse(Condition := converted, Message := 'Did not report ULINT to TIME conversion was prevented');

TEST_FINISHED();
END_METHOD

METHOD PUBLIC Check_ULINT_TO_TIME_Max
VAR
	value : ULINT := DatatypeLimits.MAX_VALUE_OF_ULINT_WHICH_CAN_BE_HELD_IN_A_TIME;
	actual : TIME;
	converted : BOOL;
	equal : BOOL;
END_VAR
TEST('Check_ULINT_TO_TIME_Max');

// @TEST-RUN
converted := TryConvert_ULINT_TO_Destination(value, actual);
equal := actual = ULINT_TO_TIME(value);

// @TEST-ASSERT
AssertTrue(Condition := equal, Message := 'Did not convert ULINT to TIME correctly');
AssertTrue(Condition := converted, Message := 'Did not report ULINT to TIME conversion was successful');

TEST_FINISHED();
END_METHOD

METHOD PUBLIC Check_ULINT_TO_TOD_Min
VAR
	value : ULINT := DatatypeLimits.ULINT_MIN_VALUE;
	actual : TOD;
	converted : BOOL;
	equal : BOOL;
END_VAR
TEST('Check_ULINT_TO_TOD_Min');

// @TEST-RUN
converted := TryConvert_ULINT_TO_Destination(value, actual);
equal := actual = ULINT_TO_TOD(value);

// @TEST-ASSERT
AssertTrue(Condition := equal, Message := 'Did not convert ULINT to TOD correctly');
AssertTrue(Condition := converted, Message := 'Did not report ULINT to TOD conversion was successful');

TEST_FINISHED();
END_METHOD

METHOD PUBLIC Check_ULINT_TO_TOD_TooHigh
VAR
	value : ULINT := DatatypeLimits.ULINT_MAX_VALUE;
	actual : TOD;
	converted : BOOL;
END_VAR
TEST('Check_ULINT_TO_TOD_TooHigh');

// @TEST-RUN
converted := TryConvert_ULINT_TO_Destination(value, actual);

// @TEST-ASSERT
AssertFalse(Condition := converted, Message := 'Did not report ULINT to TOD conversion was prevented');

TEST_FINISHED();
END_METHOD

METHOD PUBLIC Check_ULINT_TO_TOD_Max
VAR
	value : ULINT := DatatypeLimits.MAX_VALUE_OF_ULINT_WHICH_CAN_BE_HELD_IN_A_TOD;
	actual : TOD;
	converted : BOOL;
	equal : BOOL;
END_VAR
TEST('Check_ULINT_TO_TOD_Max');

// @TEST-RUN
converted := TryConvert_ULINT_TO_Destination(value, actual);
equal := actual = ULINT_TO_TOD(value);

// @TEST-ASSERT
AssertTrue(Condition := equal, Message := 'Did not convert ULINT to TOD correctly');
AssertTrue(Condition := converted, Message := 'Did not report ULINT to TOD conversion was successful');

TEST_FINISHED();
END_METHOD

METHOD PUBLIC Check_ULINT_TO_UDINT_Min
VAR
	value : ULINT := DatatypeLimits.ULINT_MIN_VALUE;
	actual : UDINT;
	converted : BOOL;
	equal : BOOL;
END_VAR
TEST('Check_ULINT_TO_UDINT_Min');

// @TEST-RUN
converted := TryConvert_ULINT_TO_Destination(value, actual);
equal := actual = ULINT_TO_UDINT(value);

// @TEST-ASSERT
AssertTrue(Condition := equal, Message := 'Did not convert ULINT to UDINT correctly');
AssertTrue(Condition := converted, Message := 'Did not report ULINT to UDINT conversion was successful');

TEST_FINISHED();
END_METHOD

METHOD PUBLIC Check_ULINT_TO_UDINT_TooHigh
VAR
	value : ULINT := DatatypeLimits.ULINT_MAX_VALUE;
	actual : UDINT;
	converted : BOOL;
END_VAR
TEST('Check_ULINT_TO_UDINT_TooHigh');

// @TEST-RUN
converted := TryConvert_ULINT_TO_Destination(value, actual);

// @TEST-ASSERT
AssertFalse(Condition := converted, Message := 'Did not report ULINT to UDINT conversion was prevented');

TEST_FINISHED();
END_METHOD

METHOD PUBLIC Check_ULINT_TO_UDINT_Max
VAR
	value : ULINT := DatatypeLimits.MAX_VALUE_OF_ULINT_WHICH_CAN_BE_HELD_IN_A_UDINT;
	actual : UDINT;
	converted : BOOL;
	equal : BOOL;
END_VAR
TEST('Check_ULINT_TO_UDINT_Max');

// @TEST-RUN
converted := TryConvert_ULINT_TO_Destination(value, actual);
equal := actual = ULINT_TO_UDINT(value);

// @TEST-ASSERT
AssertTrue(Condition := equal, Message := 'Did not convert ULINT to UDINT correctly');
AssertTrue(Condition := converted, Message := 'Did not report ULINT to UDINT conversion was successful');

TEST_FINISHED();
END_METHOD

METHOD PUBLIC Check_ULINT_TO_UINT_Min
VAR
	value : ULINT := DatatypeLimits.ULINT_MIN_VALUE;
	actual : UINT;
	converted : BOOL;
	equal : BOOL;
END_VAR
TEST('Check_ULINT_TO_UINT_Min');

// @TEST-RUN
converted := TryConvert_ULINT_TO_Destination(value, actual);
equal := actual = ULINT_TO_UINT(value);

// @TEST-ASSERT
AssertTrue(Condition := equal, Message := 'Did not convert ULINT to UINT correctly');
AssertTrue(Condition := converted, Message := 'Did not report ULINT to UINT conversion was successful');

TEST_FINISHED();
END_METHOD

METHOD PUBLIC Check_ULINT_TO_UINT_TooHigh
VAR
	value : ULINT := DatatypeLimits.ULINT_MAX_VALUE;
	actual : UINT;
	converted : BOOL;
END_VAR
TEST('Check_ULINT_TO_UINT_TooHigh');

// @TEST-RUN
converted := TryConvert_ULINT_TO_Destination(value, actual);

// @TEST-ASSERT
AssertFalse(Condition := converted, Message := 'Did not report ULINT to UINT conversion was prevented');

TEST_FINISHED();
END_METHOD

METHOD PUBLIC Check_ULINT_TO_UINT_Max
VAR
	value : ULINT := DatatypeLimits.MAX_VALUE_OF_ULINT_WHICH_CAN_BE_HELD_IN_A_UINT;
	actual : UINT;
	converted : BOOL;
	equal : BOOL;
END_VAR
TEST('Check_ULINT_TO_UINT_Max');

// @TEST-RUN
converted := TryConvert_ULINT_TO_Destination(value, actual);
equal := actual = ULINT_TO_UINT(value);

// @TEST-ASSERT
AssertTrue(Condition := equal, Message := 'Did not convert ULINT to UINT correctly');
AssertTrue(Condition := converted, Message := 'Did not report ULINT to UINT conversion was successful');

TEST_FINISHED();
END_METHOD

METHOD PUBLIC Check_ULINT_TO_ULINT_Min
VAR
	value : ULINT := DatatypeLimits.ULINT_MIN_VALUE;
	actual : ULINT;
	converted : BOOL;
	equal : BOOL;
END_VAR
TEST('Check_ULINT_TO_ULINT_Min');

// @TEST-RUN
converted := TryConvert_ULINT_TO_Destination(value, actual);
equal := actual = value;

// @TEST-ASSERT
AssertTrue(Condition := equal, Message := 'Did not convert ULINT to ULINT correctly');
AssertTrue(Condition := converted, Message := 'Did not report ULINT to ULINT conversion was successful');

TEST_FINISHED();
END_METHOD

METHOD PUBLIC Check_ULINT_TO_ULINT_Max
VAR
	value : ULINT := DatatypeLimits.ULINT_MAX_VALUE;
	actual : ULINT;
	converted : BOOL;
	equal : BOOL;
END_VAR
TEST('Check_ULINT_TO_ULINT_Max');

// @TEST-RUN
converted := TryConvert_ULINT_TO_Destination(value, actual);
equal := actual = value;

// @TEST-ASSERT
AssertTrue(Condition := equal, Message := 'Did not convert ULINT to ULINT correctly');
AssertTrue(Condition := converted, Message := 'Did not report ULINT to ULINT conversion was successful');

TEST_FINISHED();
END_METHOD

METHOD PUBLIC Check_ULINT_TO_USINT_Min
VAR
	value : ULINT := DatatypeLimits.ULINT_MIN_VALUE;
	actual : USINT;
	converted : BOOL;
	equal : BOOL;
END_VAR
TEST('Check_ULINT_TO_USINT_Min');

// @TEST-RUN
converted := TryConvert_ULINT_TO_Destination(value, actual);
equal := actual = ULINT_TO_USINT(value);

// @TEST-ASSERT
AssertTrue(Condition := equal, Message := 'Did not convert ULINT to USINT correctly');
AssertTrue(Condition := converted, Message := 'Did not report ULINT to USINT conversion was successful');

TEST_FINISHED();
END_METHOD

METHOD PUBLIC Check_ULINT_TO_USINT_TooHigh
VAR
	value : ULINT := DatatypeLimits.ULINT_MAX_VALUE;
	actual : USINT;
	converted : BOOL;
END_VAR
TEST('Check_ULINT_TO_USINT_TooHigh');

// @TEST-RUN
converted := TryConvert_ULINT_TO_Destination(value, actual);

// @TEST-ASSERT
AssertFalse(Condition := converted, Message := 'Did not report ULINT to USINT conversion was prevented');

TEST_FINISHED();
END_METHOD

METHOD PUBLIC Check_ULINT_TO_USINT_Max
VAR
	value : ULINT := DatatypeLimits.MAX_VALUE_OF_ULINT_WHICH_CAN_BE_HELD_IN_A_USINT;
	actual : USINT;
	converted : BOOL;
	equal : BOOL;
END_VAR
TEST('Check_ULINT_TO_USINT_Max');

// @TEST-RUN
converted := TryConvert_ULINT_TO_Destination(value, actual);
equal := actual = ULINT_TO_USINT(value);

// @TEST-ASSERT
AssertTrue(Condition := equal, Message := 'Did not convert ULINT to USINT correctly');
AssertTrue(Condition := converted, Message := 'Did not report ULINT to USINT conversion was successful');

TEST_FINISHED();
END_METHOD

METHOD PUBLIC Check_ULINT_TO_WORD_Min
VAR
	value : ULINT := DatatypeLimits.ULINT_MIN_VALUE;
	actual : WORD;
	converted : BOOL;
	equal : BOOL;
END_VAR
TEST('Check_ULINT_TO_WORD_Min');

// @TEST-RUN
converted := TryConvert_ULINT_TO_Destination(value, actual);
equal := actual = ULINT_TO_WORD(value);

// @TEST-ASSERT
AssertTrue(Condition := equal, Message := 'Did not convert ULINT to WORD correctly');
AssertTrue(Condition := converted, Message := 'Did not report ULINT to WORD conversion was successful');

TEST_FINISHED();
END_METHOD

METHOD PUBLIC Check_ULINT_TO_WORD_TooHigh
VAR
	value : ULINT := DatatypeLimits.ULINT_MAX_VALUE;
	actual : WORD;
	converted : BOOL;
END_VAR
TEST('Check_ULINT_TO_WORD_TooHigh');

// @TEST-RUN
converted := TryConvert_ULINT_TO_Destination(value, actual);

// @TEST-ASSERT
AssertFalse(Condition := converted, Message := 'Did not report ULINT to WORD conversion was prevented');

TEST_FINISHED();
END_METHOD

METHOD PUBLIC Check_ULINT_TO_WORD_Max
VAR
	value : ULINT := DatatypeLimits.MAX_VALUE_OF_ULINT_WHICH_CAN_BE_HELD_IN_A_WORD;
	actual : WORD;
	converted : BOOL;
	equal : BOOL;
END_VAR
TEST('Check_ULINT_TO_WORD_Max');

// @TEST-RUN
converted := TryConvert_ULINT_TO_Destination(value, actual);
equal := actual = ULINT_TO_WORD(value);

// @TEST-ASSERT
AssertTrue(Condition := equal, Message := 'Did not convert ULINT to WORD correctly');
AssertTrue(Condition := converted, Message := 'Did not report ULINT to WORD conversion was successful');

TEST_FINISHED();
END_METHOD

END_FUNCTION_BLOCK

// ---- Tests/REAL_TO_TestSuite.TcPOU
FUNCTION_BLOCK PUBLIC REAL_TO_TestSuite EXTENDS TcUnit.FB_TestSuite
VAR
END_VAR

Check_REAL_TO_BOOL_Max();
Check_REAL_TO_BOOL_Min();
Check_REAL_TO_BYTE_Max();
Check_REAL_TO_BYTE_Min();
Check_REAL_TO_BYTE_TooHigh();
Check_REAL_TO_BYTE_TooLow();
Check_REAL_TO_WORD_Max();
Check_REAL_TO_WORD_Min();
Check_REAL_TO_WORD_TooHigh();
Check_REAL_TO_WORD_TooLow();
Check_REAL_TO_DWORD_Max();
Check_REAL_TO_DWORD_Min();
Check_REAL_TO_DWORD_TooHigh();
Check_REAL_TO_DWORD_TooLow();
Check_REAL_TO_LWORD_Max();
Check_REAL_TO_LWORD_Min();
Check_REAL_TO_LWORD_TooHigh();
Check_REAL_TO_LWORD_TooLow();
Check_REAL_TO_SINT_Max();
Check_REAL_TO_SINT_Min();
Check_REAL_TO_SINT_TooHigh();
Check_REAL_TO_SINT_TooLow();
Check_REAL_TO_INT_Max();
Check_REAL_TO_INT_Min();
Check_REAL_TO_INT_TooHigh();
Check_REAL_TO_INT_TooLow();
Check_REAL_TO_DINT_Max();
Check_REAL_TO_DINT_Min();
Check_REAL_TO_DINT_TooHigh();
Check_REAL_TO_DINT_TooLow();
Check_REAL_TO_LINT_Max();
Check_REAL_TO_LINT_Min();
Check_REAL_TO_LINT_TooHigh();
Check_REAL_TO_LINT_TooLow();
Check_REAL_TO_USINT_Max();
Check_REAL_TO_USINT_Min();
Check_REAL_TO_USINT_TooHigh();
Check_REAL_TO_USINT_TooLow();
Check_REAL_TO_UINT_Max();
Check_REAL_TO_UINT_Min();
Check_REAL_TO_UINT_TooHigh();
Check_REAL_TO_UINT_TooLow();
Check_REAL_TO_UDINT_Max();
Check_REAL_TO_UDINT_Min();
Check_REAL_TO_UDINT_TooHigh();
Check_REAL_TO_UDINT_TooLow();
Check_REAL_TO_ULINT_Max();
Check_REAL_TO_ULINT_Min();
Check_REAL_TO_ULINT_TooHigh();
Check_REAL_TO_ULINT_TooLow();
Check_REAL_TO_REAL_Max();
Check_REAL_TO_REAL_Min();
Check_REAL_TO_LREAL_Max();
Check_REAL_TO_LREAL_Min();
Check_REAL_TO_TIME_Max();
Check_REAL_TO_TIME_Min();
Check_REAL_TO_TIME_TooHigh();
Check_REAL_TO_TIME_TooLow();
Check_REAL_TO_TOD_Max();
Check_REAL_TO_TOD_Min();
Check_REAL_TO_TOD_TooHigh();
Check_REAL_TO_TOD_TooLow();
Check_REAL_TO_DATE_Max();
Check_REAL_TO_DATE_Min();
Check_REAL_TO_DATE_TooHigh();
Check_REAL_TO_DATE_TooLow();
Check_REAL_TO_DT_Max();
Check_REAL_TO_DT_Min();
Check_REAL_TO_DT_TooHigh();
Check_REAL_TO_DT_TooLow();
Check_REAL_TO_STRING_Max();
Check_REAL_TO_STRING_Min();

METHOD PUBLIC Check_REAL_TO_BOOL_Min
VAR
	value : REAL := DatatypeLimits.REAL_MIN_VALUE;
	actual : BOOL;
	converted : BOOL;
	equal : BOOL;
END_VAR
TEST('Check_REAL_TO_BOOL_Min');

// @TEST-RUN
converted := TryConvert_REAL_TO_Destination(value, actual);
equal := actual = REAL_TO_BOOL(value);

// @TEST-ASSERT
AssertTrue(Condition := equal, Message := 'Did not convert REAL to BOOL correctly');
AssertTrue(Condition := converted, Message := 'Did not report REAL to BOOL conversion was successful');

TEST_FINISHED();
END_METHOD

METHOD PUBLIC Check_REAL_TO_BOOL_Max
VAR
	value : REAL := DatatypeLimits.REAL_MAX_VALUE;
	actual : BOOL;
	converted : BOOL;
	equal : BOOL;
END_VAR
TEST('Check_REAL_TO_BOOL_Max');

// @TEST-RUN
converted := TryConvert_REAL_TO_Destination(value, actual);
equal := actual = REAL_TO_BOOL(value);

// @TEST-ASSERT
AssertTrue(Condition := equal, Message := 'Did not convert REAL to BOOL correctly');
AssertTrue(Condition := converted, Message := 'Did not report REAL to BOOL conversion was successful');

TEST_FINISHED();
END_METHOD

METHOD PUBLIC Check_REAL_TO_BYTE_Min
VAR
	value : REAL := DatatypeLimits.MIN_VALUE_OF_REAL_WHICH_CAN_BE_HELD_IN_A_BYTE;
	actual : BYTE;
	converted : BOOL;
	equal : BOOL;
END_VAR
TEST('Check_REAL_TO_BYTE_Min');

// @TEST-RUN
converted := TryConvert_REAL_TO_Destination(value, actual);
equal := actual = REAL_TO_BYTE(value);

// @TEST-ASSERT
AssertTrue(Condition := equal, Message := 'Did not convert REAL to BYTE correctly');
AssertTrue(Condition := converted, Message := 'Did not report REAL to BYTE conversion was successful');

TEST_FINISHED();
END_METHOD

METHOD PUBLIC Check_REAL_TO_BYTE_TooHigh
VAR
	value : REAL := DatatypeLimits.REAL_MAX_VALUE;
	actual : BYTE;
	converted : BOOL;
END_VAR
TEST('Check_REAL_TO_BYTE_TooHigh');

// @TEST-RUN
converted := TryConvert_REAL_TO_Destination(value, actual);

// @TEST-ASSERT
AssertFalse(Condition := converted, Message := 'Did not report REAL to BYTE conversion was prevented');

TEST_FINISHED();
END_METHOD

METHOD PUBLIC Check_REAL_TO_BYTE_TooLow
VAR
	value : REAL := DatatypeLimits.REAL_MIN_VALUE;
	actual : BYTE;
	converted : BOOL;
END_VAR
TEST('Check_REAL_TO_BYTE_TooLow');

// @TEST-RUN
converted := TryConvert_REAL_TO_Destination(value, actual);

// @TEST-ASSERT
AssertFalse(Condition := converted, Message := 'Did not report REAL to BYTE conversion was prevented');

TEST_FINISHED();
END_METHOD

METHOD PUBLIC Check_REAL_TO_BYTE_Max
VAR
	value : REAL := DatatypeLimits.MAX_VALUE_OF_REAL_WHICH_CAN_BE_HELD_IN_A_BYTE;
	actual : BYTE;
	converted : BOOL;
	equal : BOOL;
END_VAR
TEST('Check_REAL_TO_BYTE_Max');

// @TEST-RUN
converted := TryConvert_REAL_TO_Destination(value, actual);
equal := actual = REAL_TO_BYTE(value);

// @TEST-ASSERT
AssertTrue(Condition := equal, Message := 'Did not convert REAL to BYTE correctly');
AssertTrue(Condition := converted, Message := 'Did not report REAL to BYTE conversion was successful');

TEST_FINISHED();
END_METHOD

METHOD PUBLIC Check_REAL_TO_DATE_Min
VAR
	value : REAL := DatatypeLimits.MIN_VALUE_OF_REAL_WHICH_CAN_BE_HELD_IN_A_DATE;
	actual : DATE;
	converted : BOOL;
	equal : BOOL;
END_VAR
TEST('Check_REAL_TO_DATE_Min');

// @TEST-RUN
converted := TryConvert_REAL_TO_Destination(value, actual);
equal := actual = REAL_TO_DATE(value);

// @TEST-ASSERT
AssertTrue(Condition := equal, Message := 'Did not convert REAL to DATE correctly');
AssertTrue(Condition := converted, Message := 'Did not report REAL to DATE conversion was successful');

TEST_FINISHED();
END_METHOD

METHOD PUBLIC Check_REAL_TO_DATE_TooHigh
VAR
	value : REAL := DatatypeLimits.REAL_MAX_VALUE;
	actual : DATE;
	converted : BOOL;
END_VAR
TEST('Check_REAL_TO_DATE_TooHigh');

// @TEST-RUN
converted := TryConvert_REAL_TO_Destination(value, actual);

// @TEST-ASSERT
AssertFalse(Condition := converted, Message := 'Did not report REAL to DATE conversion was prevented');

TEST_FINISHED();
END_METHOD

METHOD PUBLIC Check_REAL_TO_DATE_TooLow
VAR
	value : REAL := DatatypeLimits.REAL_MIN_VALUE;
	actual : DATE;
	converted : BOOL;
END_VAR
TEST('Check_REAL_TO_DATE_TooLow');

// @TEST-RUN
converted := TryConvert_REAL_TO_Destination(value, actual);

// @TEST-ASSERT
AssertFalse(Condition := converted, Message := 'Did not report REAL to DATE conversion was prevented');

TEST_FINISHED();
END_METHOD

METHOD PUBLIC Check_REAL_TO_DATE_Max
VAR
	value : REAL := DatatypeLimits.MAX_VALUE_OF_REAL_WHICH_CAN_BE_HELD_IN_A_DATE;
	actual : DATE;
	converted : BOOL;
	equal : BOOL;
END_VAR
TEST('Check_REAL_TO_DATE_Max');

// @TEST-RUN
converted := TryConvert_REAL_TO_Destination(value, actual);
equal := actual = REAL_TO_DATE(value);

// @TEST-ASSERT
AssertTrue(Condition := equal, Message := 'Did not convert REAL to DATE correctly');
AssertTrue(Condition := converted, Message := 'Did not report REAL to DATE conversion was successful');

TEST_FINISHED();
END_METHOD

METHOD PUBLIC Check_REAL_TO_DINT_Min
VAR
	value : REAL := DatatypeLimits.MIN_VALUE_OF_REAL_WHICH_CAN_BE_HELD_IN_A_DINT;
	actual : DINT;
	converted : BOOL;
	equal : BOOL;
END_VAR
TEST('Check_REAL_TO_DINT_Min');

// @TEST-RUN
converted := TryConvert_REAL_TO_Destination(value, actual);
equal := actual = REAL_TO_DINT(value);

// @TEST-ASSERT
AssertTrue(Condition := equal, Message := 'Did not convert REAL to DINT correctly');
AssertTrue(Condition := converted, Message := 'Did not report REAL to DINT conversion was successful');

TEST_FINISHED();
END_METHOD

METHOD PUBLIC Check_REAL_TO_DINT_TooHigh
VAR
	value : REAL := DatatypeLimits.REAL_MAX_VALUE;
	actual : DINT;
	converted : BOOL;
END_VAR
TEST('Check_REAL_TO_DINT_TooHigh');

// @TEST-RUN
converted := TryConvert_REAL_TO_Destination(value, actual);

// @TEST-ASSERT
AssertFalse(Condition := converted, Message := 'Did not report REAL to DINT conversion was prevented');

TEST_FINISHED();
END_METHOD

METHOD PUBLIC Check_REAL_TO_DINT_TooLow
VAR
	value : REAL := DatatypeLimits.REAL_MIN_VALUE;
	actual : DINT;
	converted : BOOL;
END_VAR
TEST('Check_REAL_TO_DINT_TooLow');

// @TEST-RUN
converted := TryConvert_REAL_TO_Destination(value, actual);

// @TEST-ASSERT
AssertFalse(Condition := converted, Message := 'Did not report REAL to DINT conversion was prevented');

TEST_FINISHED();
END_METHOD

METHOD PUBLIC Check_REAL_TO_DINT_Max
VAR
	value : REAL := DatatypeLimits.MAX_VALUE_OF_REAL_WHICH_CAN_BE_HELD_IN_A_DINT;
	actual : DINT;
	converted : BOOL;
	equal : BOOL;
END_VAR
TEST('Check_REAL_TO_DINT_Max');

// @TEST-RUN
converted := TryConvert_REAL_TO_Destination(value, actual);
equal := actual = REAL_TO_DINT(value);

// @TEST-ASSERT
AssertTrue(Condition := equal, Message := 'Did not convert REAL to DINT correctly');
AssertTrue(Condition := converted, Message := 'Did not report REAL to DINT conversion was successful');

TEST_FINISHED();
END_METHOD

METHOD PUBLIC Check_REAL_TO_DT_Min
VAR
	value : REAL := DatatypeLimits.MIN_VALUE_OF_REAL_WHICH_CAN_BE_HELD_IN_A_DT;
	actual : DT;
	converted : BOOL;
	equal : BOOL;
END_VAR
TEST('Check_REAL_TO_DT_Min');

// @TEST-RUN
converted := TryConvert_REAL_TO_Destination(value, actual);
equal := actual = REAL_TO_DT(value);

// @TEST-ASSERT
AssertTrue(Condition := equal, Message := 'Did not convert REAL to DT correctly');
AssertTrue(Condition := converted, Message := 'Did not report REAL to DT conversion was successful');

TEST_FINISHED();
END_METHOD

METHOD PUBLIC Check_REAL_TO_DT_TooHigh
VAR
	value : REAL := DatatypeLimits.REAL_MAX_VALUE;
	actual : DT;
	converted : BOOL;
END_VAR
TEST('Check_REAL_TO_DT_TooHigh');

// @TEST-RUN
converted := TryConvert_REAL_TO_Destination(value, actual);

// @TEST-ASSERT
AssertFalse(Condition := converted, Message := 'Did not report REAL to DT conversion was prevented');

TEST_FINISHED();
END_METHOD

METHOD PUBLIC Check_REAL_TO_DT_TooLow
VAR
	value : REAL := DatatypeLimits.REAL_MIN_VALUE;
	actual : DT;
	converted : BOOL;
END_VAR
TEST('Check_REAL_TO_DT_TooLow');

// @TEST-RUN
converted := TryConvert_REAL_TO_Destination(value, actual);

// @TEST-ASSERT
AssertFalse(Condition := converted, Message := 'Did not report REAL to DT conversion was prevented');

TEST_FINISHED();
END_METHOD

METHOD PUBLIC Check_REAL_TO_DT_Max
VAR
	value : REAL := DatatypeLimits.MAX_VALUE_OF_REAL_WHICH_CAN_BE_HELD_IN_A_DT;
	actual : DT;
	converted : BOOL;
	equal : BOOL;
END_VAR
TEST('Check_REAL_TO_DT_Max');

// @TEST-RUN
converted := TryConvert_REAL_TO_Destination(value, actual);
equal := actual = REAL_TO_DT(value);

// @TEST-ASSERT
AssertTrue(Condition := equal, Message := 'Did not convert REAL to DT correctly');
AssertTrue(Condition := converted, Message := 'Did not report REAL to DT conversion was successful');

TEST_FINISHED();
END_METHOD

METHOD PUBLIC Check_REAL_TO_DWORD_Min
VAR
	value : REAL := DatatypeLimits.MIN_VALUE_OF_REAL_WHICH_CAN_BE_HELD_IN_A_DWORD;
	actual : DWORD;
	converted : BOOL;
	equal : BOOL;
END_VAR
TEST('Check_REAL_TO_DWORD_Min');

// @TEST-RUN
converted := TryConvert_REAL_TO_Destination(value, actual);
equal := actual = REAL_TO_DWORD(value);

// @TEST-ASSERT
AssertTrue(Condition := equal, Message := 'Did not convert REAL to DWORD correctly');
AssertTrue(Condition := converted, Message := 'Did not report REAL to DWORD conversion was successful');

TEST_FINISHED();
END_METHOD

METHOD PUBLIC Check_REAL_TO_DWORD_TooHigh
VAR
	value : REAL := DatatypeLimits.REAL_MAX_VALUE;
	actual : DWORD;
	converted : BOOL;
END_VAR
TEST('Check_REAL_TO_DWORD_TooHigh');

// @TEST-RUN
converted := TryConvert_REAL_TO_Destination(value, actual);

// @TEST-ASSERT
AssertFalse(Condition := converted, Message := 'Did not report REAL to DWORD conversion was prevented');

TEST_FINISHED();
END_METHOD

METHOD PUBLIC Check_REAL_TO_DWORD_TooLow
VAR
	value : REAL := DatatypeLimits.REAL_MIN_VALUE;
	actual : DWORD;
	converted : BOOL;
END_VAR
TEST('Check_REAL_TO_DWORD_TooLow');

// @TEST-RUN
converted := TryConvert_REAL_TO_Destination(value, actual);

// @TEST-ASSERT
AssertFalse(Condition := converted, Message := 'Did not report REAL to DWORD conversion was prevented');

TEST_FINISHED();
END_METHOD

METHOD PUBLIC Check_REAL_TO_DWORD_Max
VAR
	value : REAL := DatatypeLimits.MAX_VALUE_OF_REAL_WHICH_CAN_BE_HELD_IN_A_DWORD;
	actual : DWORD;
	converted : BOOL;
	equal : BOOL;
END_VAR
TEST('Check_REAL_TO_DWORD_Max');

// @TEST-RUN
converted := TryConvert_REAL_TO_Destination(value, actual);
equal := actual = REAL_TO_DWORD(value);

// @TEST-ASSERT
AssertTrue(Condition := equal, Message := 'Did not convert REAL to DWORD correctly');
AssertTrue(Condition := converted, Message := 'Did not report REAL to DWORD conversion was successful');

TEST_FINISHED();
END_METHOD

METHOD PUBLIC Check_REAL_TO_INT_Min
VAR
	value : REAL := DatatypeLimits.MIN_VALUE_OF_REAL_WHICH_CAN_BE_HELD_IN_A_INT;
	actual : INT;
	converted : BOOL;
	equal : BOOL;
END_VAR
TEST('Check_REAL_TO_INT_Min');

// @TEST-RUN
converted := TryConvert_REAL_TO_Destination(value, actual);
equal := actual = REAL_TO_INT(value);

// @TEST-ASSERT
AssertTrue(Condition := equal, Message := 'Did not convert REAL to INT correctly');
AssertTrue(Condition := converted, Message := 'Did not report REAL to INT conversion was successful');

TEST_FINISHED();
END_METHOD

METHOD PUBLIC Check_REAL_TO_INT_TooHigh
VAR
	value : REAL := DatatypeLimits.REAL_MAX_VALUE;
	actual : INT;
	converted : BOOL;
END_VAR
TEST('Check_REAL_TO_INT_TooHigh');

// @TEST-RUN
converted := TryConvert_REAL_TO_Destination(value, actual);

// @TEST-ASSERT
AssertFalse(Condition := converted, Message := 'Did not report REAL to INT conversion was prevented');

TEST_FINISHED();
END_METHOD

METHOD PUBLIC Check_REAL_TO_INT_TooLow
VAR
	value : REAL := DatatypeLimits.REAL_MIN_VALUE;
	actual : INT;
	converted : BOOL;
END_VAR
TEST('Check_REAL_TO_INT_TooLow');

// @TEST-RUN
converted := TryConvert_REAL_TO_Destination(value, actual);

// @TEST-ASSERT
AssertFalse(Condition := converted, Message := 'Did not report REAL to INT conversion was prevented');

TEST_FINISHED();
END_METHOD

METHOD PUBLIC Check_REAL_TO_INT_Max
VAR
	value : REAL := DatatypeLimits.MAX_VALUE_OF_REAL_WHICH_CAN_BE_HELD_IN_A_INT;
	actual : INT;
	converted : BOOL;
	equal : BOOL;
END_VAR
TEST('Check_REAL_TO_INT_Max');

// @TEST-RUN
converted := TryConvert_REAL_TO_Destination(value, actual);
equal := actual = REAL_TO_INT(value);

// @TEST-ASSERT
AssertTrue(Condition := equal, Message := 'Did not convert REAL to INT correctly');
AssertTrue(Condition := converted, Message := 'Did not report REAL to INT conversion was successful');

TEST_FINISHED();
END_METHOD

METHOD PUBLIC Check_REAL_TO_LINT_Min
VAR
	value : REAL := DatatypeLimits.MIN_VALUE_OF_REAL_WHICH_CAN_BE_HELD_IN_A_LINT;
	actual : LINT;
	converted : BOOL;
	equal : BOOL;
END_VAR
TEST('Check_REAL_TO_LINT_Min');

// @TEST-RUN
converted := TryConvert_REAL_TO_Destination(value, actual);
equal := actual = REAL_TO_LINT(value);

// @TEST-ASSERT
AssertTrue(Condition := equal, Message := 'Did not convert REAL to LINT correctly');
AssertTrue(Condition := converted, Message := 'Did not report REAL to LINT conversion was successful');

TEST_FINISHED();
END_METHOD

METHOD PUBLIC Check_REAL_TO_LINT_TooHigh
VAR
	value : REAL := DatatypeLimits.REAL_MAX_VALUE;
	actual : LINT;
	converted : BOOL;
END_VAR
TEST('Check_REAL_TO_LINT_TooHigh');

// @TEST-RUN
converted := TryConvert_REAL_TO_Destination(value, actual);

// @TEST-ASSERT
AssertFalse(Condition := converted, Message := 'Did not report REAL to LINT conversion was prevented');

TEST_FINISHED();
END_METHOD

METHOD PUBLIC Check_REAL_TO_LINT_TooLow
VAR
	value : REAL := DatatypeLimits.REAL_MIN_VALUE;
	actual : LINT;
	converted : BOOL;
END_VAR
TEST('Check_REAL_TO_LINT_TooLow');

// @TEST-RUN
converted := TryConvert_REAL_TO_Destination(value, actual);

// @TEST-ASSERT
AssertFalse(Condition := converted, Message := 'Did not report REAL to LINT conversion was prevented');

TEST_FINISHED();
END_METHOD

METHOD PUBLIC Check_REAL_TO_LINT_Max
VAR
	value : REAL := DatatypeLimits.MAX_VALUE_OF_REAL_WHICH_CAN_BE_HELD_IN_A_LINT;
	actual : LINT;
	converted : BOOL;
	equal : BOOL;
END_VAR
TEST('Check_REAL_TO_LINT_Max');

// @TEST-RUN
converted := TryConvert_REAL_TO_Destination(value, actual);
equal := actual = REAL_TO_LINT(value);

// @TEST-ASSERT
AssertTrue(Condition := equal, Message := 'Did not convert REAL to LINT correctly');
AssertTrue(Condition := converted, Message := 'Did not report REAL to LINT conversion was successful');

TEST_FINISHED();
END_METHOD

METHOD PUBLIC Check_REAL_TO_LREAL_Min
VAR
	value : REAL := DatatypeLimits.REAL_MIN_VALUE;
	actual : LREAL;
	converted : BOOL;
	equal : BOOL;
END_VAR
TEST('Check_REAL_TO_LREAL_Min');

// @TEST-RUN
converted := TryConvert_REAL_TO_Destination(value, actual);
equal := actual = REAL_TO_LREAL(value);

// @TEST-ASSERT
AssertTrue(Condition := equal, Message := 'Did not convert REAL to LREAL correctly');
AssertTrue(Condition := converted, Message := 'Did not report REAL to LREAL conversion was successful');

TEST_FINISHED();
END_METHOD

METHOD PUBLIC Check_REAL_TO_LREAL_Max
VAR
	value : REAL := DatatypeLimits.REAL_MAX_VALUE;
	actual : LREAL;
	converted : BOOL;
	equal : BOOL;
END_VAR
TEST('Check_REAL_TO_LREAL_Max');

// @TEST-RUN
converted := TryConvert_REAL_TO_Destination(value, actual);
equal := actual = REAL_TO_LREAL(value);

// @TEST-ASSERT
AssertTrue(Condition := equal, Message := 'Did not convert REAL to LREAL correctly');
AssertTrue(Condition := converted, Message := 'Did not report REAL to LREAL conversion was successful');

TEST_FINISHED();
END_METHOD

METHOD PUBLIC Check_REAL_TO_LWORD_Min
VAR
	value : REAL := DatatypeLimits.MIN_VALUE_OF_REAL_WHICH_CAN_BE_HELD_IN_A_LWORD;
	actual : LWORD;
	converted : BOOL;
	equal : BOOL;
END_VAR
TEST('Check_REAL_TO_LWORD_Min');

// @TEST-RUN
converted := TryConvert_REAL_TO_Destination(value, actual);
equal := actual = REAL_TO_LWORD(value);

// @TEST-ASSERT
AssertTrue(Condition := equal, Message := 'Did not convert REAL to LWORD correctly');
AssertTrue(Condition := converted, Message := 'Did not report REAL to LWORD conversion was successful');

TEST_FINISHED();
END_METHOD

METHOD PUBLIC Check_REAL_TO_LWORD_TooHigh
VAR
	value : REAL := DatatypeLimits.REAL_MAX_VALUE;
	actual : LWORD;
	converted : BOOL;
END_VAR
TEST('Check_REAL_TO_LWORD_TooHigh');

// @TEST-RUN
converted := TryConvert_REAL_TO_Destination(value, actual);

// @TEST-ASSERT
AssertFalse(Condition := converted, Message := 'Did not report REAL to LWORD conversion was prevented');

TEST_FINISHED();
END_METHOD

METHOD PUBLIC Check_REAL_TO_LWORD_TooLow
VAR
	value : REAL := DatatypeLimits.REAL_MIN_VALUE;
	actual : LWORD;
	converted : BOOL;
END_VAR
TEST('Check_REAL_TO_LWORD_TooLow');

// @TEST-RUN
converted := TryConvert_REAL_TO_Destination(value, actual);

// @TEST-ASSERT
AssertFalse(Condition := converted, Message := 'Did not report REAL to LWORD conversion was prevented');

TEST_FINISHED();
END_METHOD

METHOD PUBLIC Check_REAL_TO_LWORD_Max
VAR
	value : REAL := DatatypeLimits.MAX_VALUE_OF_REAL_WHICH_CAN_BE_HELD_IN_A_LWORD;
	actual : LWORD;
	converted : BOOL;
	equal : BOOL;
END_VAR
TEST('Check_REAL_TO_LWORD_Max');

// @TEST-RUN
converted := TryConvert_REAL_TO_Destination(value, actual);
equal := actual = REAL_TO_LWORD(value);

// @TEST-ASSERT
AssertTrue(Condition := equal, Message := 'Did not convert REAL to LWORD correctly');
AssertTrue(Condition := converted, Message := 'Did not report REAL to LWORD conversion was successful');

TEST_FINISHED();
END_METHOD

METHOD PUBLIC Check_REAL_TO_REAL_Min
VAR
	value : REAL := DatatypeLimits.REAL_MIN_VALUE;
	actual : REAL;
	converted : BOOL;
	equal : BOOL;
END_VAR
TEST('Check_REAL_TO_REAL_Min');

// @TEST-RUN
converted := TryConvert_REAL_TO_Destination(value, actual);
equal := actual = value;

// @TEST-ASSERT
AssertTrue(Condition := equal, Message := 'Did not convert REAL to REAL correctly');
AssertTrue(Condition := converted, Message := 'Did not report REAL to REAL conversion was successful');

TEST_FINISHED();
END_METHOD

METHOD PUBLIC Check_REAL_TO_REAL_Max
VAR
	value : REAL := DatatypeLimits.REAL_MAX_VALUE;
	actual : REAL;
	converted : BOOL;
	equal : BOOL;
END_VAR
TEST('Check_REAL_TO_REAL_Max');

// @TEST-RUN
converted := TryConvert_REAL_TO_Destination(value, actual);
equal := actual = value;

// @TEST-ASSERT
AssertTrue(Condition := equal, Message := 'Did not convert REAL to REAL correctly');
AssertTrue(Condition := converted, Message := 'Did not report REAL to REAL conversion was successful');

TEST_FINISHED();
END_METHOD

METHOD PUBLIC Check_REAL_TO_SINT_Min
VAR
	value : REAL := DatatypeLimits.MIN_VALUE_OF_REAL_WHICH_CAN_BE_HELD_IN_A_SINT;
	actual : SINT;
	converted : BOOL;
	equal : BOOL;
END_VAR
TEST('Check_REAL_TO_SINT_Min');

// @TEST-RUN
converted := TryConvert_REAL_TO_Destination(value, actual);
equal := actual = REAL_TO_SINT(value);

// @TEST-ASSERT
AssertTrue(Condition := equal, Message := 'Did not convert REAL to SINT correctly');
AssertTrue(Condition := converted, Message := 'Did not report REAL to SINT conversion was successful');

TEST_FINISHED();
END_METHOD

METHOD PUBLIC Check_REAL_TO_SINT_TooHigh
VAR
	value : REAL := DatatypeLimits.REAL_MAX_VALUE;
	actual : SINT;
	converted : BOOL;
END_VAR
TEST('Check_REAL_TO_SINT_TooHigh');

// @TEST-RUN
converted := TryConvert_REAL_TO_Destination(value, actual);

// @TEST-ASSERT
AssertFalse(Condition := converted, Message := 'Did not report REAL to SINT conversion was prevented');

TEST_FINISHED();
END_METHOD

METHOD PUBLIC Check_REAL_TO_SINT_TooLow
VAR
	value : REAL := DatatypeLimits.REAL_MIN_VALUE;
	actual : SINT;
	converted : BOOL;
END_VAR
TEST('Check_REAL_TO_SINT_TooLow');

// @TEST-RUN
converted := TryConvert_REAL_TO_Destination(value, actual);

// @TEST-ASSERT
AssertFalse(Condition := converted, Message := 'Did not report REAL to SINT conversion was prevented');

TEST_FINISHED();
END_METHOD

METHOD PUBLIC Check_REAL_TO_SINT_Max
VAR
	value : REAL := DatatypeLimits.MAX_VALUE_OF_REAL_WHICH_CAN_BE_HELD_IN_A_SINT;
	actual : SINT;
	converted : BOOL;
	equal : BOOL;
END_VAR
TEST('Check_REAL_TO_SINT_Max');

// @TEST-RUN
converted := TryConvert_REAL_TO_Destination(value, actual);
equal := actual = REAL_TO_SINT(value);

// @TEST-ASSERT
AssertTrue(Condition := equal, Message := 'Did not convert REAL to SINT correctly');
AssertTrue(Condition := converted, Message := 'Did not report REAL to SINT conversion was successful');

TEST_FINISHED();
END_METHOD

METHOD PUBLIC Check_REAL_TO_STRING_Min
VAR
	value : REAL := DatatypeLimits.REAL_MIN_VALUE;
	actual : STRING;
	converted : BOOL;
	equal : BOOL;
END_VAR
TEST('Check_REAL_TO_STRING_Min');

// @TEST-RUN
converted := TryConvert_REAL_TO_Destination(value, actual);
equal := actual = REAL_TO_STRING(value);

// @TEST-ASSERT
AssertTrue(Condition := equal, Message := 'Did not convert REAL to STRING correctly');
AssertTrue(Condition := converted, Message := 'Did not report REAL to STRING conversion was successful');

TEST_FINISHED();
END_METHOD

METHOD PUBLIC Check_REAL_TO_STRING_Max
VAR
	value : REAL := DatatypeLimits.REAL_MAX_VALUE;
	actual : STRING;
	converted : BOOL;
	equal : BOOL;
END_VAR
TEST('Check_REAL_TO_STRING_Max');

// @TEST-RUN
converted := TryConvert_REAL_TO_Destination(value, actual);
equal := actual = REAL_TO_STRING(value);

// @TEST-ASSERT
AssertTrue(Condition := equal, Message := 'Did not convert REAL to STRING correctly');
AssertTrue(Condition := converted, Message := 'Did not report REAL to STRING conversion was successful');

TEST_FINISHED();
END_METHOD

METHOD PUBLIC Check_REAL_TO_TIME_Min
VAR
	value : REAL := DatatypeLimits.MIN_VALUE_OF_REAL_WHICH_CAN_BE_HELD_IN_A_TIME;
	actual : TIME;
	converted : BOOL;
	equal : BOOL;
END_VAR
TEST('Check_REAL_TO_TIME_Min');

// @TEST-RUN
converted := TryConvert_REAL_TO_Destination(value, actual);
equal := actual = REAL_TO_TIME(value);

// @TEST-ASSERT
AssertTrue(Condition := equal, Message := 'Did not convert REAL to TIME correctly');
AssertTrue(Condition := converted, Message := 'Did not report REAL to TIME conversion was successful');

TEST_FINISHED();
END_METHOD

METHOD PUBLIC Check_REAL_TO_TIME_TooHigh
VAR
	value : REAL := DatatypeLimits.REAL_MAX_VALUE;
	actual : TIME;
	converted : BOOL;
END_VAR
TEST('Check_REAL_TO_TIME_TooHigh');

// @TEST-RUN
converted := TryConvert_REAL_TO_Destination(value, actual);

// @TEST-ASSERT
AssertFalse(Condition := converted, Message := 'Did not report REAL to TIME conversion was prevented');

TEST_FINISHED();
END_METHOD

METHOD PUBLIC Check_REAL_TO_TIME_TooLow
VAR
	value : REAL := DatatypeLimits.REAL_MIN_VALUE;
	actual : TIME;
	converted : BOOL;
END_VAR
TEST('Check_REAL_TO_TIME_TooLow');

// @TEST-RUN
converted := TryConvert_REAL_TO_Destination(value, actual);

// @TEST-ASSERT
AssertFalse(Condition := converted, Message := 'Did not report REAL to TIME conversion was prevented');

TEST_FINISHED();
END_METHOD

METHOD PUBLIC Check_REAL_TO_TIME_Max
VAR
	value : REAL := DatatypeLimits.MAX_VALUE_OF_REAL_WHICH_CAN_BE_HELD_IN_A_TIME;
	actual : TIME;
	converted : BOOL;
	equal : BOOL;
END_VAR
TEST('Check_REAL_TO_TIME_Max');

// @TEST-RUN
converted := TryConvert_REAL_TO_Destination(value, actual);
equal := actual = REAL_TO_TIME(value);

// @TEST-ASSERT
AssertTrue(Condition := equal, Message := 'Did not convert REAL to TIME correctly');
AssertTrue(Condition := converted, Message := 'Did not report REAL to TIME conversion was successful');

TEST_FINISHED();
END_METHOD

METHOD PUBLIC Check_REAL_TO_TOD_Min
VAR
	value : REAL := DatatypeLimits.MIN_VALUE_OF_REAL_WHICH_CAN_BE_HELD_IN_A_TOD;
	actual : TOD;
	converted : BOOL;
	equal : BOOL;
END_VAR
TEST('Check_REAL_TO_TOD_Min');

// @TEST-RUN
converted := TryConvert_REAL_TO_Destination(value, actual);
equal := actual = REAL_TO_TOD(value);

// @TEST-ASSERT
AssertTrue(Condition := equal, Message := 'Did not convert REAL to TOD correctly');
AssertTrue(Condition := converted, Message := 'Did not report REAL to TOD conversion was successful');

TEST_FINISHED();
END_METHOD

METHOD PUBLIC Check_REAL_TO_TOD_TooHigh
VAR
	value : REAL := DatatypeLimits.REAL_MAX_VALUE;
	actual : TOD;
	converted : BOOL;
END_VAR
TEST('Check_REAL_TO_TOD_TooHigh');

// @TEST-RUN
converted := TryConvert_REAL_TO_Destination(value, actual);

// @TEST-ASSERT
AssertFalse(Condition := converted, Message := 'Did not report REAL to TOD conversion was prevented');

TEST_FINISHED();
END_METHOD

METHOD PUBLIC Check_REAL_TO_TOD_TooLow
VAR
	value : REAL := DatatypeLimits.REAL_MIN_VALUE;
	actual : TOD;
	converted : BOOL;
END_VAR
TEST('Check_REAL_TO_TOD_TooLow');

// @TEST-RUN
converted := TryConvert_REAL_TO_Destination(value, actual);

// @TEST-ASSERT
AssertFalse(Condition := converted, Message := 'Did not report REAL to TOD conversion was prevented');

TEST_FINISHED();
END_METHOD

METHOD PUBLIC Check_REAL_TO_TOD_Max
VAR
	value : REAL := DatatypeLimits.MAX_VALUE_OF_REAL_WHICH_CAN_BE_HELD_IN_A_TOD;
	actual : TOD;
	converted : BOOL;
	equal : BOOL;
END_VAR
TEST('Check_REAL_TO_TOD_Max');

// @TEST-RUN
converted := TryConvert_REAL_TO_Destination(value, actual);
equal := actual = REAL_TO_TOD(value);

// @TEST-ASSERT
AssertTrue(Condition := equal, Message := 'Did not convert REAL to TOD correctly');
AssertTrue(Condition := converted, Message := 'Did not report REAL to TOD conversion was successful');

TEST_FINISHED();
END_METHOD

METHOD PUBLIC Check_REAL_TO_UDINT_Min
VAR
	value : REAL := DatatypeLimits.MIN_VALUE_OF_REAL_WHICH_CAN_BE_HELD_IN_A_UDINT;
	actual : UDINT;
	converted : BOOL;
	equal : BOOL;
END_VAR
TEST('Check_REAL_TO_UDINT_Min');

// @TEST-RUN
converted := TryConvert_REAL_TO_Destination(value, actual);
equal := actual = REAL_TO_UDINT(value);

// @TEST-ASSERT
AssertTrue(Condition := equal, Message := 'Did not convert REAL to UDINT correctly');
AssertTrue(Condition := converted, Message := 'Did not report REAL to UDINT conversion was successful');

TEST_FINISHED();
END_METHOD

METHOD PUBLIC Check_REAL_TO_UDINT_TooHigh
VAR
	value : REAL := DatatypeLimits.REAL_MAX_VALUE;
	actual : UDINT;
	converted : BOOL;
END_VAR
TEST('Check_REAL_TO_UDINT_TooHigh');

// @TEST-RUN
converted := TryConvert_REAL_TO_Destination(value, actual);

// @TEST-ASSERT
AssertFalse(Condition := converted, Message := 'Did not report REAL to UDINT conversion was prevented');

TEST_FINISHED();
END_METHOD

METHOD PUBLIC Check_REAL_TO_UDINT_TooLow
VAR
	value : REAL := DatatypeLimits.REAL_MIN_VALUE;
	actual : UDINT;
	converted : BOOL;
END_VAR
TEST('Check_REAL_TO_UDINT_TooLow');

// @TEST-RUN
converted := TryConvert_REAL_TO_Destination(value, actual);

// @TEST-ASSERT
AssertFalse(Condition := converted, Message := 'Did not report REAL to UDINT conversion was prevented');

TEST_FINISHED();
END_METHOD

METHOD PUBLIC Check_REAL_TO_UDINT_Max
VAR
	value : REAL := DatatypeLimits.MAX_VALUE_OF_REAL_WHICH_CAN_BE_HELD_IN_A_UDINT;
	actual : UDINT;
	converted : BOOL;
	equal : BOOL;
END_VAR
TEST('Check_REAL_TO_UDINT_Max');

// @TEST-RUN
converted := TryConvert_REAL_TO_Destination(value, actual);
equal := actual = REAL_TO_UDINT(value);

// @TEST-ASSERT
AssertTrue(Condition := equal, Message := 'Did not convert REAL to UDINT correctly');
AssertTrue(Condition := converted, Message := 'Did not report REAL to UDINT conversion was successful');

TEST_FINISHED();
END_METHOD

METHOD PUBLIC Check_REAL_TO_UINT_Min
VAR
	value : REAL := DatatypeLimits.MIN_VALUE_OF_REAL_WHICH_CAN_BE_HELD_IN_A_UINT;
	actual : UINT;
	converted : BOOL;
	equal : BOOL;
END_VAR
TEST('Check_REAL_TO_UINT_Min');

// @TEST-RUN
converted := TryConvert_REAL_TO_Destination(value, actual);
equal := actual = REAL_TO_UINT(value);

// @TEST-ASSERT
AssertTrue(Condition := equal, Message := 'Did not convert REAL to UINT correctly');
AssertTrue(Condition := converted, Message := 'Did not report REAL to UINT conversion was successful');

TEST_FINISHED();
END_METHOD

METHOD PUBLIC Check_REAL_TO_UINT_TooHigh
VAR
	value : REAL := DatatypeLimits.REAL_MAX_VALUE;
	actual : UINT;
	converted : BOOL;
END_VAR
TEST('Check_REAL_TO_UINT_TooHigh');

// @TEST-RUN
converted := TryConvert_REAL_TO_Destination(value, actual);

// @TEST-ASSERT
AssertFalse(Condition := converted, Message := 'Did not report REAL to UINT conversion was prevented');

TEST_FINISHED();
END_METHOD

METHOD PUBLIC Check_REAL_TO_UINT_TooLow
VAR
	value : REAL := DatatypeLimits.REAL_MIN_VALUE;
	actual : UINT;
	converted : BOOL;
END_VAR
TEST('Check_REAL_TO_UINT_TooLow');

// @TEST-RUN
converted := TryConvert_REAL_TO_Destination(value, actual);

// @TEST-ASSERT
AssertFalse(Condition := converted, Message := 'Did not report REAL to UINT conversion was prevented');

TEST_FINISHED();
END_METHOD

METHOD PUBLIC Check_REAL_TO_UINT_Max
VAR
	value : REAL := DatatypeLimits.MAX_VALUE_OF_REAL_WHICH_CAN_BE_HELD_IN_A_UINT;
	actual : UINT;
	converted : BOOL;
	equal : BOOL;
END_VAR
TEST('Check_REAL_TO_UINT_Max');

// @TEST-RUN
converted := TryConvert_REAL_TO_Destination(value, actual);
equal := actual = REAL_TO_UINT(value);

// @TEST-ASSERT
AssertTrue(Condition := equal, Message := 'Did not convert REAL to UINT correctly');
AssertTrue(Condition := converted, Message := 'Did not report REAL to UINT conversion was successful');

TEST_FINISHED();
END_METHOD

METHOD PUBLIC Check_REAL_TO_ULINT_Min
VAR
	value : REAL := DatatypeLimits.MIN_VALUE_OF_REAL_WHICH_CAN_BE_HELD_IN_A_ULINT;
	actual : ULINT;
	converted : BOOL;
	equal : BOOL;
END_VAR
TEST('Check_REAL_TO_ULINT_Min');

// @TEST-RUN
converted := TryConvert_REAL_TO_Destination(value, actual);
equal := actual = REAL_TO_ULINT(value);

// @TEST-ASSERT
AssertTrue(Condition := equal, Message := 'Did not convert REAL to ULINT correctly');
AssertTrue(Condition := converted, Message := 'Did not report REAL to ULINT conversion was successful');

TEST_FINISHED();
END_METHOD

METHOD PUBLIC Check_REAL_TO_ULINT_TooHigh
VAR
	value : REAL := DatatypeLimits.REAL_MAX_VALUE;
	actual : ULINT;
	converted : BOOL;
END_VAR
TEST('Check_REAL_TO_ULINT_TooHigh');

// @TEST-RUN
converted := TryConvert_REAL_TO_Destination(value, actual);

// @TEST-ASSERT
AssertFalse(Condition := converted, Message := 'Did not report REAL to ULINT conversion was prevented');

TEST_FINISHED();
END_METHOD

METHOD PUBLIC Check_REAL_TO_ULINT_TooLow
VAR
	value : REAL := DatatypeLimits.REAL_MIN_VALUE;
	actual : ULINT;
	converted : BOOL;
END_VAR
TEST('Check_REAL_TO_ULINT_TooLow');

// @TEST-RUN
converted := TryConvert_REAL_TO_Destination(value, actual);

// @TEST-ASSERT
AssertFalse(Condition := converted, Message := 'Did not report REAL to ULINT conversion was prevented');

TEST_FINISHED();
END_METHOD

METHOD PUBLIC Check_REAL_TO_ULINT_Max
VAR
	value : REAL := DatatypeLimits.MAX_VALUE_OF_REAL_WHICH_CAN_BE_HELD_IN_A_ULINT;
	actual : ULINT;
	converted : BOOL;
	equal : BOOL;
END_VAR
TEST('Check_REAL_TO_ULINT_Max');

// @TEST-RUN
converted := TryConvert_REAL_TO_Destination(value, actual);
equal := actual = REAL_TO_ULINT(value);

// @TEST-ASSERT
AssertTrue(Condition := equal, Message := 'Did not convert REAL to ULINT correctly');
AssertTrue(Condition := converted, Message := 'Did not report REAL to ULINT conversion was successful');

TEST_FINISHED();
END_METHOD

METHOD PUBLIC Check_REAL_TO_USINT_Min
VAR
	value : REAL := DatatypeLimits.MIN_VALUE_OF_REAL_WHICH_CAN_BE_HELD_IN_A_USINT;
	actual : USINT;
	converted : BOOL;
	equal : BOOL;
END_VAR
TEST('Check_REAL_TO_USINT_Min');

// @TEST-RUN
converted := TryConvert_REAL_TO_Destination(value, actual);
equal := actual = REAL_TO_USINT(value);

// @TEST-ASSERT
AssertTrue(Condition := equal, Message := 'Did not convert REAL to USINT correctly');
AssertTrue(Condition := converted, Message := 'Did not report REAL to USINT conversion was successful');

TEST_FINISHED();
END_METHOD

METHOD PUBLIC Check_REAL_TO_USINT_TooHigh
VAR
	value : REAL := DatatypeLimits.REAL_MAX_VALUE;
	actual : USINT;
	converted : BOOL;
END_VAR
TEST('Check_REAL_TO_USINT_TooHigh');

// @TEST-RUN
converted := TryConvert_REAL_TO_Destination(value, actual);

// @TEST-ASSERT
AssertFalse(Condition := converted, Message := 'Did not report REAL to USINT conversion was prevented');

TEST_FINISHED();
END_METHOD

METHOD PUBLIC Check_REAL_TO_USINT_TooLow
VAR
	value : REAL := DatatypeLimits.REAL_MIN_VALUE;
	actual : USINT;
	converted : BOOL;
END_VAR
TEST('Check_REAL_TO_USINT_TooLow');

// @TEST-RUN
converted := TryConvert_REAL_TO_Destination(value, actual);

// @TEST-ASSERT
AssertFalse(Condition := converted, Message := 'Did not report REAL to USINT conversion was prevented');

TEST_FINISHED();
END_METHOD

METHOD PUBLIC Check_REAL_TO_USINT_Max
VAR
	value : REAL := DatatypeLimits.MAX_VALUE_OF_REAL_WHICH_CAN_BE_HELD_IN_A_USINT;
	actual : USINT;
	converted : BOOL;
	equal : BOOL;
END_VAR
TEST('Check_REAL_TO_USINT_Max');

// @TEST-RUN
converted := TryConvert_REAL_TO_Destination(value, actual);
equal := actual = REAL_TO_USINT(value);

// @TEST-ASSERT
AssertTrue(Condition := equal, Message := 'Did not convert REAL to USINT correctly');
AssertTrue(Condition := converted, Message := 'Did not report REAL to USINT conversion was successful');

TEST_FINISHED();
END_METHOD

METHOD PUBLIC Check_REAL_TO_WORD_Min
VAR
	value : REAL := DatatypeLimits.MIN_VALUE_OF_REAL_WHICH_CAN_BE_HELD_IN_A_WORD;
	actual : WORD;
	converted : BOOL;
	equal : BOOL;
END_VAR
TEST('Check_REAL_TO_WORD_Min');

// @TEST-RUN
converted := TryConvert_REAL_TO_Destination(value, actual);
equal := actual = REAL_TO_WORD(value);

// @TEST-ASSERT
AssertTrue(Condition := equal, Message := 'Did not convert REAL to WORD correctly');
AssertTrue(Condition := converted, Message := 'Did not report REAL to WORD conversion was successful');

TEST_FINISHED();
END_METHOD

METHOD PUBLIC Check_REAL_TO_WORD_TooHigh
VAR
	value : REAL := DatatypeLimits.REAL_MAX_VALUE;
	actual : WORD;
	converted : BOOL;
END_VAR
TEST('Check_REAL_TO_WORD_TooHigh');

// @TEST-RUN
converted := TryConvert_REAL_TO_Destination(value, actual);

// @TEST-ASSERT
AssertFalse(Condition := converted, Message := 'Did not report REAL to WORD conversion was prevented');

TEST_FINISHED();
END_METHOD

METHOD PUBLIC Check_REAL_TO_WORD_TooLow
VAR
	value : REAL := DatatypeLimits.REAL_MIN_VALUE;
	actual : WORD;
	converted : BOOL;
END_VAR
TEST('Check_REAL_TO_WORD_TooLow');

// @TEST-RUN
converted := TryConvert_REAL_TO_Destination(value, actual);

// @TEST-ASSERT
AssertFalse(Condition := converted, Message := 'Did not report REAL to WORD conversion was prevented');

TEST_FINISHED();
END_METHOD

METHOD PUBLIC Check_REAL_TO_WORD_Max
VAR
	value : REAL := DatatypeLimits.MAX_VALUE_OF_REAL_WHICH_CAN_BE_HELD_IN_A_WORD;
	actual : WORD;
	converted : BOOL;
	equal : BOOL;
END_VAR
TEST('Check_REAL_TO_WORD_Max');

// @TEST-RUN
converted := TryConvert_REAL_TO_Destination(value, actual);
equal := actual = REAL_TO_WORD(value);

// @TEST-ASSERT
AssertTrue(Condition := equal, Message := 'Did not convert REAL to WORD correctly');
AssertTrue(Condition := converted, Message := 'Did not report REAL to WORD conversion was successful');

TEST_FINISHED();
END_METHOD

END_FUNCTION_BLOCK

// ---- Tests/LREAL_TO_TestSuite.TcPOU
FUNCTION_BLOCK PUBLIC LREAL_TO_TestSuite EXTENDS TcUnit.FB_TestSuite
VAR
END_VAR

Check_LREAL_TO_BOOL_Max();
Check_LREAL_TO_BOOL_Min();
Check_LREAL_TO_BYTE_Max();
Check_LREAL_TO_BYTE_Min();
Check_LREAL_TO_BYTE_TooHigh();
Check_LREAL_TO_BYTE_TooLow();
Check_LREAL_TO_WORD_Max();
Check_LREAL_TO_WORD_Min();
Check_LREAL_TO_WORD_TooHigh();
Check_LREAL_TO_WORD_TooLow();
Check_LREAL_TO_DWORD_Max();
Check_LREAL_TO_DWORD_Min();
Check_LREAL_TO_DWORD_TooHigh();
Check_LREAL_TO_DWORD_TooLow();
Check_LREAL_TO_LWORD_Max();
Check_LREAL_TO_LWORD_Min();
Check_LREAL_TO_LWORD_TooHigh();
Check_LREAL_TO_LWORD_TooLow();
Check_LREAL_TO_SINT_Max();
Check_LREAL_TO_SINT_Min();
Check_LREAL_TO_SINT_TooHigh();
Check_LREAL_TO_SINT_TooLow();
Check_LREAL_TO_INT_Max();
Check_LREAL_TO_INT_Min();
Check_LREAL_TO_INT_TooHigh();
Check_LREAL_TO_INT_TooLow();
Check_LREAL_TO_DINT_Max();
Check_LREAL_TO_DINT_Min();
Check_LREAL_TO_DINT_TooHigh();
Check_LREAL_TO_DINT_TooLow();
Check_LREAL_TO_LINT_Max();
Check_LREAL_TO_LINT_Min();
Check_LREAL_TO_LINT_TooHigh();
Check_LREAL_TO_LINT_TooLow();
Check_LREAL_TO_USINT_Max();
Check_LREAL_TO_USINT_Min();
Check_LREAL_TO_USINT_TooHigh();
Check_LREAL_TO_USINT_TooLow();
Check_LREAL_TO_UINT_Max();
Check_LREAL_TO_UINT_Min();
Check_LREAL_TO_UINT_TooHigh();
Check_LREAL_TO_UINT_TooLow();
Check_LREAL_TO_UDINT_Max();
Check_LREAL_TO_UDINT_Min();
Check_LREAL_TO_UDINT_TooHigh();
Check_LREAL_TO_UDINT_TooLow();
Check_LREAL_TO_ULINT_Max();
Check_LREAL_TO_ULINT_Min();
Check_LREAL_TO_ULINT_TooHigh();
Check_LREAL_TO_ULINT_TooLow();
Check_LREAL_TO_REAL_Max();
Check_LREAL_TO_REAL_Min();
Check_LREAL_TO_REAL_TooHigh();
Check_LREAL_TO_REAL_TooLow();
Check_LREAL_TO_LREAL_Max();
Check_LREAL_TO_LREAL_Min();
Check_LREAL_TO_TIME_Max();
Check_LREAL_TO_TIME_Min();
Check_LREAL_TO_TIME_TooHigh();
Check_LREAL_TO_TIME_TooLow();
Check_LREAL_TO_TOD_Max();
Check_LREAL_TO_TOD_Min();
Check_LREAL_TO_TOD_TooHigh();
Check_LREAL_TO_TOD_TooLow();
Check_LREAL_TO_DATE_Max();
Check_LREAL_TO_DATE_Min();
Check_LREAL_TO_DATE_TooHigh();
Check_LREAL_TO_DATE_TooLow();
Check_LREAL_TO_DT_Max();
Check_LREAL_TO_DT_Min();
Check_LREAL_TO_DT_TooHigh();
Check_LREAL_TO_DT_TooLow();
Check_LREAL_TO_STRING_Max();
Check_LREAL_TO_STRING_Min();
Check_LREAL_TO_STRING_TooHigh();
Check_LREAL_TO_STRING_TooLow();

METHOD PUBLIC Check_LREAL_TO_BOOL_Min
VAR
	value : LREAL := DatatypeLimits.LREAL_MIN_VALUE;
	actual : BOOL;
	converted : BOOL;
	equal : BOOL;
END_VAR
TEST('Check_LREAL_TO_BOOL_Min');

// @TEST-RUN
converted := TryConvert_LREAL_TO_Destination(value, actual);
equal := actual = LREAL_TO_BOOL(value);

// @TEST-ASSERT
AssertTrue(Condition := equal, Message := 'Did not convert LREAL to BOOL correctly');
AssertTrue(Condition := converted, Message := 'Did not report LREAL to BOOL conversion was successful');

TEST_FINISHED();
END_METHOD

METHOD PUBLIC Check_LREAL_TO_BOOL_Max
VAR
	value : LREAL := DatatypeLimits.LREAL_MAX_VALUE;
	actual : BOOL;
	converted : BOOL;
	equal : BOOL;
END_VAR
TEST('Check_LREAL_TO_BOOL_Max');

// @TEST-RUN
converted := TryConvert_LREAL_TO_Destination(value, actual);
equal := actual = LREAL_TO_BOOL(value);

// @TEST-ASSERT
AssertTrue(Condition := equal, Message := 'Did not convert LREAL to BOOL correctly');
AssertTrue(Condition := converted, Message := 'Did not report LREAL to BOOL conversion was successful');

TEST_FINISHED();
END_METHOD

METHOD PUBLIC Check_LREAL_TO_BYTE_Min
VAR
	value : LREAL := DatatypeLimits.MIN_VALUE_OF_LREAL_WHICH_CAN_BE_HELD_IN_A_BYTE;
	actual : BYTE;
	converted : BOOL;
	equal : BOOL;
END_VAR
TEST('Check_LREAL_TO_BYTE_Min');

// @TEST-RUN
converted := TryConvert_LREAL_TO_Destination(value, actual);
equal := actual = LREAL_TO_BYTE(value);

// @TEST-ASSERT
AssertTrue(Condition := equal, Message := 'Did not convert LREAL to BYTE correctly');
AssertTrue(Condition := converted, Message := 'Did not report LREAL to BYTE conversion was successful');

TEST_FINISHED();
END_METHOD

METHOD PUBLIC Check_LREAL_TO_BYTE_TooHigh
VAR
	value : LREAL := DatatypeLimits.LREAL_MAX_VALUE;
	actual : BYTE;
	converted : BOOL;
END_VAR
TEST('Check_LREAL_TO_BYTE_TooHigh');

// @TEST-RUN
converted := TryConvert_LREAL_TO_Destination(value, actual);

// @TEST-ASSERT
AssertFalse(Condition := converted, Message := 'Did not report LREAL to BYTE conversion was prevented');

TEST_FINISHED();
END_METHOD

METHOD PUBLIC Check_LREAL_TO_BYTE_TooLow
VAR
	value : LREAL := DatatypeLimits.LREAL_MIN_VALUE;
	actual : BYTE;
	converted : BOOL;
END_VAR
TEST('Check_LREAL_TO_BYTE_TooLow');

// @TEST-RUN
converted := TryConvert_LREAL_TO_Destination(value, actual);

// @TEST-ASSERT
AssertFalse(Condition := converted, Message := 'Did not report LREAL to BYTE conversion was prevented');

TEST_FINISHED();
END_METHOD

METHOD PUBLIC Check_LREAL_TO_BYTE_Max
VAR
	value : LREAL := DatatypeLimits.MAX_VALUE_OF_LREAL_WHICH_CAN_BE_HELD_IN_A_BYTE;
	actual : BYTE;
	converted : BOOL;
	equal : BOOL;
END_VAR
TEST('Check_LREAL_TO_BYTE_Max');

// @TEST-RUN
converted := TryConvert_LREAL_TO_Destination(value, actual);
equal := actual = LREAL_TO_BYTE(value);

// @TEST-ASSERT
AssertTrue(Condition := equal, Message := 'Did not convert LREAL to BYTE correctly');
AssertTrue(Condition := converted, Message := 'Did not report LREAL to BYTE conversion was successful');

TEST_FINISHED();
END_METHOD

METHOD PUBLIC Check_LREAL_TO_DATE_Min
VAR
	value : LREAL := DatatypeLimits.MIN_VALUE_OF_LREAL_WHICH_CAN_BE_HELD_IN_A_DATE;
	actual : DATE;
	converted : BOOL;
	equal : BOOL;
END_VAR
TEST('Check_LREAL_TO_DATE_Min');

// @TEST-RUN
converted := TryConvert_LREAL_TO_Destination(value, actual);
equal := actual = LREAL_TO_DATE(value);

// @TEST-ASSERT
AssertTrue(Condition := equal, Message := 'Did not convert LREAL to DATE correctly');
AssertTrue(Condition := converted, Message := 'Did not report LREAL to DATE conversion was successful');

TEST_FINISHED();
END_METHOD

METHOD PUBLIC Check_LREAL_TO_DATE_TooHigh
VAR
	value : LREAL := DatatypeLimits.LREAL_MAX_VALUE;
	actual : DATE;
	converted : BOOL;
END_VAR
TEST('Check_LREAL_TO_DATE_TooHigh');

// @TEST-RUN
converted := TryConvert_LREAL_TO_Destination(value, actual);

// @TEST-ASSERT
AssertFalse(Condition := converted, Message := 'Did not report LREAL to DATE conversion was prevented');

TEST_FINISHED();
END_METHOD

METHOD PUBLIC Check_LREAL_TO_DATE_TooLow
VAR
	value : LREAL := DatatypeLimits.LREAL_MIN_VALUE;
	actual : DATE;
	converted : BOOL;
END_VAR
TEST('Check_LREAL_TO_DATE_TooLow');

// @TEST-RUN
converted := TryConvert_LREAL_TO_Destination(value, actual);

// @TEST-ASSERT
AssertFalse(Condition := converted, Message := 'Did not report LREAL to DATE conversion was prevented');

TEST_FINISHED();
END_METHOD

METHOD PUBLIC Check_LREAL_TO_DATE_Max
VAR
	value : LREAL := DatatypeLimits.MAX_VALUE_OF_LREAL_WHICH_CAN_BE_HELD_IN_A_DATE;
	actual : DATE;
	converted : BOOL;
	equal : BOOL;
END_VAR
TEST('Check_LREAL_TO_DATE_Max');

// @TEST-RUN
converted := TryConvert_LREAL_TO_Destination(value, actual);
equal := actual = LREAL_TO_DATE(value);

// @TEST-ASSERT
AssertTrue(Condition := equal, Message := 'Did not convert LREAL to DATE correctly');
AssertTrue(Condition := converted, Message := 'Did not report LREAL to DATE conversion was successful');

TEST_FINISHED();
END_METHOD

METHOD PUBLIC Check_LREAL_TO_DINT_Min
VAR
	value : LREAL := DatatypeLimits.MIN_VALUE_OF_LREAL_WHICH_CAN_BE_HELD_IN_A_DINT;
	actual : DINT;
	converted : BOOL;
	equal : BOOL;
END_VAR
TEST('Check_LREAL_TO_DINT_Min');

// @TEST-RUN
converted := TryConvert_LREAL_TO_Destination(value, actual);
equal := actual = LREAL_TO_DINT(value);

// @TEST-ASSERT
AssertTrue(Condition := equal, Message := 'Did not convert LREAL to DINT correctly');
AssertTrue(Condition := converted, Message := 'Did not report LREAL to DINT conversion was successful');

TEST_FINISHED();
END_METHOD

METHOD PUBLIC Check_LREAL_TO_DINT_TooHigh
VAR
	value : LREAL := DatatypeLimits.LREAL_MAX_VALUE;
	actual : DINT;
	converted : BOOL;
END_VAR
TEST('Check_LREAL_TO_DINT_TooHigh');

// @TEST-RUN
converted := TryConvert_LREAL_TO_Destination(value, actual);

// @TEST-ASSERT
AssertFalse(Condition := converted, Message := 'Did not report LREAL to DINT conversion was prevented');

TEST_FINISHED();
END_METHOD

METHOD PUBLIC Check_LREAL_TO_DINT_TooLow
VAR
	value : LREAL := DatatypeLimits.LREAL_MIN_VALUE;
	actual : DINT;
	converted : BOOL;
END_VAR
TEST('Check_LREAL_TO_DINT_TooLow');

// @TEST-RUN
converted := TryConvert_LREAL_TO_Destination(value, actual);

// @TEST-ASSERT
AssertFalse(Condition := converted, Message := 'Did not report LREAL to DINT conversion was prevented');

TEST_FINISHED();
END_METHOD

METHOD PUBLIC Check_LREAL_TO_DINT_Max
VAR
	value : LREAL := DatatypeLimits.MAX_VALUE_OF_LREAL_WHICH_CAN_BE_HELD_IN_A_DINT;
	actual : DINT;
	converted : BOOL;
	equal : BOOL;
END_VAR
TEST('Check_LREAL_TO_DINT_Max');

// @TEST-RUN
converted := TryConvert_LREAL_TO_Destination(value, actual);
equal := actual = LREAL_TO_DINT(value);

